// Trigger only a beam parameter mismatch
// Do not trip zero rate, unknown state, or debounce
PMPS_GVL.stCurrentBeamParameters := PMPS_GVL.cstFullBeam;
stBeamReq := PMPS_GVL.cstFullBeam;
stBeamReq.nTran := 0.5;
fbMiscFFO(
    fbArbiter:=fbArbiter,
    fbFFHWO:=fbFFHWO,
    stCurrentBeamReq:=stBeamReq,
    bKnownState:=TRUE,
    nTransitionID:=1,
);

fbFFHWO.EvaluateOutput();
AssertFalse(
    fbFFHWO.q_xFastFaultOut,
    'Did not fault with bad attenuator state',
);

TEST_FINISHED();
END_METHOD

METHOD TestDebounce
VAR_INST
    fbMiscFFO: FB_MiscStatesErrorFFO;
    fbArbiter: FB_Arbiter(5);
    fbFFHWO: FB_HardwareFFOutput := (bAutoReset := TRUE);
END_VAR
VAR
    nIter: DINT;
END_VAR

TEST('TestDebounce');

fbFFHWO.EvaluateOutput();
AssertTrue(
    fbFFHWO.q_xFastFaultOut,
    'Started with a fault prior to first FB run-through',
);
// Ask for full beam: there should be no faults of any kind
fbMiscFFO(
    fbArbiter:=fbArbiter,
    fbFFHWO:=fbFFHWO,
    stCurrentBeamReq:=PMPS_GVL.cstFullBeam,
    bKnownState:=TRUE,
    nTransitionID:=5,
);
fbFFHWO.EvaluateOutput();

AssertTrue(
    fbFFHWO.q_xFastFaultOut,
    'Started with a fault prior to trip checks',
);

// Trip and untrip the beam fast fault once, show no fault
TripUntrip(
    fbMiscFFO:=fbMiscFFO,
    fbArbiter:=fbArbiter,
    fbFFHWO:=fbFFHWO,
);
AssertTrue(
    fbFFHWO.q_xFastFaultOut,
    'Control group failed: one trip/untrip should not be enough to debounce',
);
// Trip and untrip the beam fast fault like 10 times, show fault
FOR nIter := 1 TO 10 DO
    TripUntrip(
        fbMiscFFO:=fbMiscFFO,
        fbArbiter:=fbArbiter,
        fbFFHWO:=fbFFHWO,
    );
END_FOR
AssertFalse(
    fbFFHWO.q_xFastFaultOut,
    'Debouncer failed to debounce',
);

TEST_FINISHED();
END_METHOD

METHOD TestTransitionState
VAR_INST
    fbMiscFFO: FB_MiscStatesErrorFFO;
    fbArbiter: FB_Arbiter(4);
    fbFFHWO: FB_HardwareFFOutput := (bAutoReset := TRUE);
END_VAR

TEST('TestTransitionState');

fbFFHWO.EvaluateOutput();
AssertTrue(
    fbFFHWO.q_xFastFaultOut,
    'Started with a fault',
);

// Trigger no faults, we're at an unknown state but it's a transition state
// Do not trip bad beam, zero rate, or debounce
fbArbiter.AddRequest(
    nReqID:=4,
    stReqBP:=PMPS_GVL.cstFullBeam,
    sDevName:='UnitTest',
);
PMPS_GVL.stCurrentBeamParameters := PMPS_GVL.cstFullBeam;
fbMiscFFO(
    fbArbiter:=fbArbiter,
    fbFFHWO:=fbFFHWO,
    stCurrentBeamReq:=PMPS_GVL.cstFullBeam,
    bKnownState:=FALSE,
    nTransitionID:=4,
);

fbFFHWO.EvaluateOutput();
AssertTrue(
    fbFFHWO.q_xFastFaultOut,
    'Faulted in unknown states even though we were moving normally',
);

TEST_FINISHED();
END_METHOD

METHOD TestUnknownState
VAR_INST
    fbMiscFFO: FB_MiscStatesErrorFFO;
    fbArbiter: FB_Arbiter(3);
    fbFFHWO: FB_HardwareFFOutput := (bAutoReset := TRUE);
END_VAR

TEST('TestUnknownState');

fbFFHWO.EvaluateOutput();
AssertTrue(
    fbFFHWO.q_xFastFaultOut,
    'Started with a fault',
);

// Trigger only an unknown states
// Do not trip bad beam, zero rate, or debounce
PMPS_GVL.stCurrentBeamParameters := PMPS_GVL.cstFullBeam;
fbMiscFFO(
    fbArbiter:=fbArbiter,
    fbFFHWO:=fbFFHWO,
    stCurrentBeamReq:=PMPS_GVL.cstFullBeam,
    bKnownState:=FALSE,
    nTransitionID:=3,
);

fbFFHWO.EvaluateOutput();
AssertFalse(
    fbFFHWO.q_xFastFaultOut,
    'Did not fault with unknown state',
);

TEST_FINISHED();
END_METHOD

METHOD TestZeroRate
VAR_INST
    fbMiscFFO: FB_MiscStatesErrorFFO;
    fbArbiter: FB_Arbiter(2);
    fbFFHWO: FB_HardwareFFOutput := (bAutoReset := TRUE);

    stNoBeam: ST_BeamParams;
END_VAR

TEST('TestBeamZeroRate');

fbFFHWO.EvaluateOutput();
AssertTrue(
    fbFFHWO.q_xFastFaultOut,
    'Started with a fault',
);

// Trigger only a zero rate
// Do not trip beam parameter mismatch, unknown state, or debounce
PMPS_GVL.stCurrentBeamParameters := stNoBeam;
fbMiscFFO(
    fbArbiter:=fbArbiter,
    fbFFHWO:=fbFFHWO,
    stCurrentBeamReq:=PMPS_GVL.cst0RateBeam,
    bKnownState:=TRUE,
    nTransitionID:=2
);

fbFFHWO.EvaluateOutput();
AssertFalse(
    fbFFHWO.q_xFastFaultOut,
    'Did not fault with zero rate',
);

TEST_FINISHED();
END_METHOD

METHOD TripUntrip
VAR_IN_OUT
    fbMiscFFO: FB_MiscStatesErrorFFO;
    fbArbiter: FB_Arbiter;
    fbFFHWO: FB_HardwareFFOutput;
END_VAR
VAR
    stBeamReq: ST_BeamParams;
END_VAR

// Use anything other than 0 rate, which is its own check
stBeamReq := PMPS_GVL.cstFullBeam;
stBeamReq.nTran := 0.5;
// Trip: too much beam!
PMPS_GVL.stCurrentBeamParameters := PMPS_GVL.cstFullBeam;
fbMiscFFO(
    fbArbiter:=fbArbiter,
    fbFFHWO:=fbFFHWO,
    stCurrentBeamReq:=stBeamReq,
    bKnownState:=TRUE,
    nTransitionID:=5,
);
fbFFHWO.EvaluateOutput();

// Untrip: correct beam!
PMPS_GVL.stCurrentBeamParameters := stBeamReq;
fbMiscFFO(
    fbArbiter:=fbArbiter,
    fbFFHWO:=fbFFHWO,
    stCurrentBeamReq:=stBeamReq,
    bKnownState:=TRUE,
    nTransitionID:=5,
);
fbFFHWO.EvaluateOutput();
END_METHOD

END_FUNCTION_BLOCK

// ---- POUs/Motion/PMPS/FB_MiscStatesErrorFFO.TcPOU
FUNCTION_BLOCK FB_MiscStatesErrorFFO
(*
    A catch-all for miscellaneous state FFOs that are not better organized elsewhere.
    Contains the following fast faults:
    - ffBeamParamsOK: trip the beam if the beam parameters are not safe enough for our current (known) state
    - ffZeroRate: trip the beam if we've asked for zero rate (as a shortcut)
    - ffUnknown: trip the beam if we're at an unknown state and our transition id is not asserted.
    - ffDebounce: trip the beam (no autoreset) if ffBeamParamsOK fast faults fault on and off multiple times too quickly.
      This solves an issue where ffBeamParamsOK might solve its own problem and creating a blinking fast fault issue.

    The inputs are mostly outputs of non-pmps function blocks and heavily-reused info like state details.
*)
VAR_IN_OUT
    // The arbiter to request beam states from
    fbArbiter: FB_Arbiter;
    // The fast fault output to fault to
    fbFFHWO: FB_HardwareFFOutput;
END_VAR
VAR_INPUT
    // A name to link to these fast faults
    sDeviceName: STRING;
    // Current requested beam details: either a known state or the transition beam
    stCurrentBeamReq: ST_BeamParams;
    // TRUE if we're at a known state (doesn't matter which)
    bKnownState: BOOL;
    // Lookup ID of the transition beam
    nTransitionID: DWORD;
    // Set me true to prevent any ffos from occuring
    bMaintenanceMode : BOOL;
END_VAR
VAR_OUTPUT
END_VAR
VAR CONSTANT
    // Number of consecutive trips before we debounce
    nMaxTrips: UINT := 5;
    // Decrease trip count by 1 after this much time has passed
    tTripReset: TIME := T#1s;
END_VAR
VAR
    // If the beam parameters are wrong, it is a fault! This encompasses all unknown arbiter-related errors.
    ffBeamParamsOk: FB_FastFault;
    // If we asked for zero rate (NC or SC) then we can cut the beam early. This is somewhat redundant.
    ffZeroRate: FB_FastFault;
    // Trip the beam for unknown state
    ffUnknown: FB_FastFault;
    // Trip the beam (no autoreset) if ffBeamParamsOK faults/resets multiple times too quickly.
    ffDebounce: FB_FastFault;

    // Number of consecutive trips so far
    nTripCount: UINT;
    // Increase by 1 whenever there is a fault (rising edge)
    ftTripCount: F_TRIG;
    // Decrease trip count by 1 each timeout
    tonTripCount: TON;
    // TRUE on only the first cycle
    bFirstCycle: BOOL := TRUE;
END_VAR


ffBeamParamsOk(
    i_xOK:=F_SafeBPCompare(PMPS_GVL.stCurrentBeamParameters, stCurrentBeamReq) OR bMaintenanceMode,
    i_xAutoReset:=TRUE,
    i_DevName:=sDeviceName,
    i_Desc:='Beam parameter mismatch',
    i_TypeCode:=E_MotionFFType.BP_MISMATCH,
    io_fbFFHWO:=fbFFHWO);

CASE PMPS_GVL.stCurrentBeamParameters.nMachineMode OF
    // NC mode
    1: ffZeroRate.i_xOK := stCurrentBeamReq.nRate > 0;
    // SC mode
    2: ffZeroRate.i_xOK := stCurrentBeamReq.nBCRange > 0;
ELSE
    // Ambiguous or new mode
    ffZeroRate.i_xOK := stCurrentBeamReq.nRate > 0 AND stCurrentBeamReq.nBCRange > 0;
END_CASE

ffZeroRate.i_xOK := ffZeroRate.i_xOK OR bMaintenanceMode;

ffZeroRate(
    i_xAutoReset := TRUE,
    i_DevName := sDeviceName,
    i_Desc := 'Device requesting zero rate',
    i_TypeCode := E_MotionFFType.ZERO_RATE,
    io_fbFFHWO := fbFFHWO,
);

ffUnknown(
    i_xOK := bknownState OR fbArbiter.CheckRequestInPool(nReqID:=nTransitionID) OR bMaintenanceMode,
    i_xAutoReset := TRUE,
    i_DevName := sDeviceName,
    i_Desc := 'Unknown position between moves',
    i_TypeCode := E_MotionFFType.NOT_A_STATE,
    io_fbFFHWO := fbFFHWO,
);

ftTripCount(CLK:=ffBeamParamsOk.i_xOK);

IF ftTripCount.Q THEN
    nTripCount := MIN(nTripCount + 1, 5);
END_IF

tonTripCount(
    IN:=NOT tonTripCount.Q,
    PT:=tTripReset,
);
IF tonTripCount.Q AND nTripCount > 0 THEN
    nTripCount := nTripCount - 1;
END_IF

// This is required for non-autoresetting FBs to come up in a beam permitted state
ffDebounce.i_xReset := bFirstCycle OR nTripCount=0;
ffDebounce(
    i_xOK := nTripCount < 5 OR bMaintenanceMode,
    i_DevName := sDeviceName,
    i_Desc := 'Tripped beam parameter mismatch off/on too many times, hold off',
    i_TypeCode := E_MotionFFType.TOO_MANY_TRIPS,
    io_fbFFHWO := fbFFHWO,
);
bFirstCycle := FALSE;

END_FUNCTION_BLOCK

// ---- Tests/FB_MotionBPTM_Test.TcPOU
FUNCTION_BLOCK FB_MotionBPTM_Test EXTENDS TcUnit.FB_TestSuite
(*
    Test the functionality of the motion bptm,
    Which is just a bptm wrapped up with a set of n motors.
    We're basically just making sure that we push the done button at the appropriate time.
    Direct tests of BPTM itself are reserved for the pmps library.

    The BPTM takes care of these executions across multiple cycles,
    so these tests must implement timeouts.
*)
VAR
    astMotionStage: ARRAY[1..MotionConstants.MAX_STATE_MOTORS] OF ST_MotionStage;
    stGoal1: ST_DbStateParams;
    stGoal2: ST_DbStateParams;
    stTrans: ST_DbStateParams;
    stNoBeam: ST_BeamParams;
END_VAR


stGoal1.stBeamParams := PMPS_GVL.cstFullBeam;
stGoal1.nRequestAssertionID := 1;
stGoal1.sPmpsState := 'stGoal1';
stGoal2.stBeamParams := PMPS_GVL.cstFullBeam;
stGoal2.stBeamParams.nTran := 0.5;
stGoal2.nRequestAssertionID := 2;
stGoal2.sPmpsState := 'stGoal2';
stTrans.stBeamParams := PMPS_GVL.cst0RateBeam;
stTrans.nRequestAssertionID := 3;
stTrans.sPmpsState := 'stTrans';

// Just put a blanket global no beam so these won't wait for any changes ever
PMPS_GVL.stCurrentBeamParameters := stNoBeam;
TestInit();
Test3dMove();
TestNoMove();
TestCount();
TestToggle();

METHOD AssertInPool
VAR_IN_OUT
    fbArbiter: FB_Arbiter;
    stDbStateParams: ST_DbStateParams;
END_VAR
VAR_INPUT
    bInPool: BOOL;
    sContext: STRING;
END_VAR

IF bInPool THEN
    AssertTrue(
        fbArbiter.CheckRequestInPool(stDbStateParams.nRequestAssertionID),
        CONCAT(CONCAT(stDbStateParams.sPmpsState, ' Beam parameters were not in the pool '), sContext),
    );
ELSE
    AssertFalse(
        fbArbiter.CheckRequestInPool(stDbStateParams.nRequestAssertionID),
        CONCAT(CONCAT(stDbStateParams.sPmpsState, ' Beam parameters unexpectedly found in the pool '), sContext),
    );
END_IF
END_METHOD

METHOD SetMotorDone
VAR_INPUT
END_VAR

// Force post-move state
astMotionStage[1].bBusy := FALSE;
astMotionStage[1].bDone := TRUE;
astMotionStage[2].bBusy := FALSE;
astMotionStage[2].bDone := TRUE;
astMotionStage[3].bBusy := FALSE;
astMotionStage[3].bDone := TRUE;
END_METHOD

METHOD SetMotorMoving
VAR_INPUT
END_VAR

// Force a moving but not done state
astMotionStage[1].bBusy := TRUE;
astMotionStage[1].bDone := FALSE;
astMotionStage[2].bBusy := TRUE;
astMotionStage[2].bDone := FALSE;
astMotionStage[3].bBusy := TRUE;
astMotionStage[3].bDone := FALSE;
END_METHOD

METHOD SetMotorStartup
VAR_INPUT
END_VAR

// Force some sort of default looking state
astMotionStage[1].bBusy := FALSE;
astMotionStage[1].bDone := FALSE;
astMotionStage[2].bBusy := FALSE;
astMotionStage[2].bDone := FALSE;
astMotionStage[3].bBusy := FALSE;
astMotionStage[3].bDone := FALSE;
END_METHOD

METHOD Test3dMove : BOOL
(*
    Can we safely do a 3d move?
*)
VAR_INST
    fbBptm: FB_MotionBPTM;
    fbArbiter: FB_Arbiter(2);
    fbFFHWO: FB_HardwareFFOutput := (bAutoReset := TRUE);
    fbSubSysIO : FB_DummyArbIO;

    nState: UINT;
    tonTimer: TON;
END_VAR

TEST('Test3DMove');

tonTimer(
    IN:=TRUE,
    PT:=T#5s,
);
IF tonTimer.Q THEN
    nState := 4;
END_IF

CASE nState OF
    0:
        // Establish baseline at Goal1
        SetMotorStartup();
        fbBptm(
            astMotionStage:=astMotionStage,
            fbArbiter:=fbArbiter,
            fbFFHWO:=fbFFHWO,
            stGoalParams:=stGoal1,
            stTransParams:=stTrans,
            nActiveMotorCount:=3,
            bEnable:=TRUE,
            bAtState:=TRUE,
        );
        IF fbBptm.bDone THEN
            nState := 1;
        END_IF
    1:
        // Request a move
        SetMotorStartup();
        fbBptm(
            astMotionStage:=astMotionStage,
            fbArbiter:=fbArbiter,
            fbFFHWO:=fbFFHWO,
            stGoalParams:=stGoal2,
            stTransParams:=stTrans,
            nActiveMotorCount:=3,
            bEnable:=TRUE,
            bAtState:=FALSE,
        );
        IF fbBptm.bTransitionAuthorized THEN
            // We should have transition and goal 2 asserts in
            AssertInPool(fbArbiter, stGoal1, FALSE, 'with trans auth');
            AssertInPool(fbArbiter, stGoal2, TRUE, 'with trans auth');
            AssertInPool(fbArbiter, stTrans, TRUE, 'with trans auth');
            nState := 2;
        END_IF
    2:
        // Simulate a move
        SetMotorMoving();
        fbBptm(
            astMotionStage:=astMotionStage,
            fbArbiter:=fbArbiter,
            fbFFHWO:=fbFFHWO,
            stGoalParams:=stGoal2,
            stTransParams:=stTrans,
            nActiveMotorCount:=3,
            bEnable:=TRUE,
            bAtState:=FALSE,
        );
        // Same situation as before
        AssertInPool(fbArbiter, stGoal1, FALSE, 'after move started');
        AssertInPool(fbArbiter, stGoal2, TRUE, 'after move started');
        AssertInPool(fbArbiter, stTrans, TRUE, 'after move started');
        nState := 3;
    3:
        // Move is done
        SetMotorDone();
        fbBptm(
            astMotionStage:=astMotionStage,
            fbArbiter:=fbArbiter,
            fbFFHWO:=fbFFHWO,
            stGoalParams:=stGoal2,
            stTransParams:=stTrans,
            nActiveMotorCount:=3,
            bEnable:=TRUE,
            bAtState:=TRUE,
        );
        IF fbBptm.bDone THEN
            // Dropped the transition assert
            AssertInPool(fbArbiter, stGoal1, FALSE, 'with move complete');
            AssertInPool(fbArbiter, stGoal2, TRUE, 'with move complete');
            AssertInPool(fbArbiter, stTrans, FALSE, 'with move complete');
            nState := 4;
        END_IF
    4:
        AssertFalse(
            tonTimer.Q,
            'Timeout in test',
        );
        TEST_FINISHED();
END_CASE

fbSubSysIO(
    LA:=fbArbiter,
    FFO:=fbFFHWO,
);
END_METHOD

METHOD TestCount
(*
    FB Should just error out if we forgot to give a count
*)
VAR_INST
    fbBptm: FB_MotionBPTM;
    fbArbiter: FB_Arbiter(1);
    fbFFHWO: FB_HardwareFFOutput := (bAutoReset := TRUE);

    tonWait: TON;
END_VAR
TEST('TestCount');

SetMotorStartup();
fbBptm(
    astMotionStage:=astMotionStage,
    fbArbiter:=fbArbiter,
    fbFFHWO:=fbFFHWO,
    stGoalParams:=stGoal1,
    stTransParams:=stTrans,
    bEnable:=True,
    bAtState:=True,
);
AssertTrue(
    fbBptm.bMotorCountError,
    'Did not properly error on missing motor count',
);

tonWait(
    IN:=TRUE,
    PT:=T#1s,
);
IF tonWait.Q THEN
    // Should have no arbiter activity at all
    AssertInPool(fbArbiter, stGoal1, FALSE, 'with bad count');
    AssertInPool(fbArbiter, stGoal2, FALSE, 'with bad count');
    AssertInPool(fbArbiter, stTrans, FALSE, 'with bad count');

    TEST_FINISHED();
END_IF
END_METHOD

METHOD TestInit : BOOL
(*
    If we initialize with still motors, do we get an arbiter request at the current goal? Hopefully we do.
*)
VAR_INST
    fbBptm: FB_MotionBPTM;
    fbArbiter: FB_Arbiter(1);
    fbFFHWO: FB_HardwareFFOutput := (bAutoReset := TRUE);
    fbSubSysIO : FB_DummyArbIO;

    tonTimer: TON;
END_VAR

TEST('TestInit');

SetMotorStartup();
fbBptm(
    astMotionStage:=astMotionStage,
    fbArbiter:=fbArbiter,
    fbFFHWO:=fbFFHWO,
    stGoalParams:=stGoal1,
    stTransParams:=stTrans,
    nActiveMotorCount:=3,
    bEnable:=True,
    bAtState:=True,
);
fbSubSysIO(
    LA:=fbArbiter,
    FFO:=fbFFHWO,
);

tonTimer(
    IN:=TRUE,
    PT:=T#5s,
);
IF tonTimer.Q OR fbBptm.bDone THEN
    AssertFalse(
        tonTimer.Q,
        'Timeout in test',
    );
    // We should have a request in the pool for goal 1 but not for transition
    // If no request are in the pool, we may come up in a no protection state!
    // If both requests are in the pool, we may come up in a too much blocking beam state!
    AssertInPool(fbArbiter, stGoal1, TRUE, 'at startup');
    AssertInPool(fbArbiter, stTrans, FALSE, 'at startup');

    TEST_FINISHED();
END_IF
END_METHOD

METHOD TestNoMove
(*
    In place transitions should work at startup and also at done positions.
*)
VAR_INST
    fbBptm: FB_MotionBPTM;
    fbArbiter: FB_Arbiter(1);
    fbFFHWO: FB_HardwareFFOutput := (bAutoReset := TRUE);
    fbSubSysIO : FB_DummyArbIO;

    nState: UINT;
    tonTimer: TON;
END_VAR

TEST('TestNoMove');

tonTimer(
    IN:=TRUE,
    PT:=T#5s,
);
IF tonTimer.Q THEN
    nState := 3;
END_IF

CASE nState OF
    0:
        SetMotorStartup();
        fbBptm(
            astMotionStage:=astMotionStage,
            fbArbiter:=fbArbiter,
            fbFFHWO:=fbFFHWO,
            stGoalParams:=stGoal1,
            stTransParams:=stTrans,
            nActiveMotorCount:=3,
            bEnable:=True,
            bAtState:=True,
        );
        IF fbBptm.bDone THEN
            nState := 1;
        END_IF
    1:
        SetMotorStartup();
        // NOTE: we kept bAtState TRUE the whole time, so this should be a completed in-place transition
        fbBptm(
            astMotionStage:=astMotionStage,
            fbArbiter:=fbArbiter,
            fbFFHWO:=fbFFHWO,
            stGoalParams:=stGoal2,
            stTransParams:=stTrans,
            nActiveMotorCount:=3,
            bEnable:=True,
            bAtState:=True,
        );
        IF fbBptm.bDone THEN
            // Only Goal2 should be in the pool
            AssertInPool(fbArbiter, stGoal1, FALSE, 'after switching goals (1)');
            AssertInPool(fbArbiter, stGoal2, TRUE, 'after switching goals (1)');
            AssertInPool(fbArbiter, stTrans, FALSE, 'after switching goals (1)');
            nState := 2;
        END_IF
    2:
        // Repeat from a done position!
        SetMotorDone();
        fbBptm(
            astMotionStage:=astMotionStage,
            fbArbiter:=fbArbiter,
            fbFFHWO:=fbFFHWO,
            stGoalParams:=stGoal1,
            stTransParams:=stTrans,
            nActiveMotorCount:=3,
            bEnable:=True,
            bAtState:=True,
        );
        IF fbBptm.bDone THEN
            // Only Goal1 should be in the pool
            AssertInPool(fbArbiter, stGoal1, TRUE, 'after switching goals (2)');
            AssertInPool(fbArbiter, stGoal2, FALSE, 'after switching goals (2)');
            AssertInPool(fbArbiter, stTrans, FALSE, 'after switching goals (2)');
            nState := 3;
        END_IF
    3:
        AssertFalse(
            tonTimer.Q,
            'Timeout in test',
        );
        TEST_FINISHED();
END_CASE

fbSubSysIO(
    LA:=fbArbiter,
    FFO:=fbFFHWO,
);
END_METHOD

METHOD TestToggle
(*
    Arbitration requests should be added to pool even if there is no transition, as case which occurs
    when a BeamParameterTransitionManager is not processed for at least one cycle without changing states
    and then reprocessed, usually when arbitration is temporarily disabled to deal with unrelated faults.
*)
VAR_INST
    fbBptm: FB_MotionBPTM;
    fbArbiter: FB_Arbiter(1);
    fbFFHWO: FB_HardwareFFOutput := (bAutoReset := TRUE);
    fbSubSysIO : FB_DummyArbIO;

    nState: UINT;
    tonTimer: TON;
END_VAR

TEST('TestToggle');

tonTimer(
    IN:=TRUE,
    PT:=T#5s,
);
IF tonTimer.Q THEN
    nState := 4;
END_IF

CASE nState OF
    0:
        SetMotorStartup();
        fbBptm(
            astMotionStage:=astMotionStage,
            fbArbiter:=fbArbiter,
            fbFFHWO:=fbFFHWO,
            stGoalParams:=stGoal1,
            stTransParams:=stTrans,
            nActiveMotorCount:=3,
            bEnable:=True,
            bAtState:=True,
        );
        IF fbBptm.bDone THEN
            nState := 1;
        END_IF
    1:
        SetMotorStartup();
        // NOTE: we kept bAtState TRUE the whole time, so this should be a completed in-place transition
        fbBptm(
            astMotionStage:=astMotionStage,
            fbArbiter:=fbArbiter,
            fbFFHWO:=fbFFHWO,
            stGoalParams:=stGoal2,
            stTransParams:=stTrans,
            nActiveMotorCount:=3,
            bEnable:=True,
            bAtState:=True,
        );
        IF fbBptm.bDone THEN
            // Only Goal2 should be in the pool
            AssertInPool(fbArbiter, stGoal1, FALSE, 'after switching goals (1)');
            AssertInPool(fbArbiter, stGoal2, TRUE, 'after switching goals (1)');
            AssertInPool(fbArbiter, stTrans, FALSE, 'after switching goals (1)');
            nState := 2;
        END_IF
    2:
        // Run disabled
        SetMotorDone();
        fbBptm(
            astMotionStage:=astMotionStage,
            fbArbiter:=fbArbiter,
            fbFFHWO:=fbFFHWO,
            stGoalParams:=stGoal2,
            stTransParams:=stTrans,
            nActiveMotorCount:=3,
            bEnable:=False,
            bAtState:=True,
        );
        IF fbBptm.bDone THEN
            // Nothing should be in the pool
            AssertInPool(fbArbiter, stGoal1, FALSE, 'after switching goals (2)');
            AssertInPool(fbArbiter, stGoal2, FALSE, 'after switching goals (2)');
            AssertInPool(fbArbiter, stTrans, FALSE, 'after switching goals (2)');
            nState := 3;
        END_IF
    3:
        // Re-enable without changing goal
        fbBptm(
            astMotionStage:=astMotionStage,
            fbArbiter:=fbArbiter,
            fbFFHWO:=fbFFHWO,
            stGoalParams:=stGoal2,
            stTransParams:=stTrans,
            nActiveMotorCount:=3,
            bEnable:=True,
            bAtState:=True,
        );
        IF fbBptm.bDone THEN
            //  Goal2 should be back in the pool
            AssertInPool(fbArbiter, stGoal1, FALSE, 'after switching goals (2)');
            AssertInPool(fbArbiter, stGoal2, TRUE, 'after switching goals (2)');
            AssertInPool(fbArbiter, stTrans, FALSE, 'after switching goals (2)');
            nState := 4;
        END_IF
    4:
        AssertFalse(
            tonTimer.Q,
            'Timeout in test',
        );
        TEST_FINISHED();
END_CASE

fbSubSysIO(
    LA:=fbArbiter,
    FFO:=fbFFHWO,
);
END_METHOD

END_FUNCTION_BLOCK

// ---- POUs/Motion/PMPS/FB_MotionBPTM.TcPOU

FUNCTION_BLOCK FB_MotionBPTM
(*
    This function block handles the beam parameter transition manager for a group of motors moving together to a destination with shared beam state.
    stGoalParams and stTransParams are required arguments and must not share IDs with other state parameters in the PLC.

    This is a building block not intended for use outside of lcls-twincat-motion.
*)
VAR_IN_OUT
    // Array of motors that will move for this beam transition
    astMotionStage: ARRAY[1..MotionConstants.MAX_STATE_MOTORS] OF ST_MotionStage;
    // The arbiter to request beam states from
    fbArbiter: FB_Arbiter;
    // The fast fault output to fault to
    fbFFHWO: FB_HardwareFFOutput;
    // The parameters we want to transition to
    stGoalParams: ST_DbStateParams;
    // The parameters we want to use during the transition
    stTransParams: ST_DbStateParams;
END_VAR
VAR_INPUT
    // The number of motors we're actually using
    nActiveMotorCount: UINT;
    // Set to TRUE to use the BPTM, FALSE to stop using the BPTM.
    bEnable: BOOL;
    // TRUE if we're at the physical state that matches the goal parameters
    bAtState: BOOL;
    // A device name to use in the GUI
    sDeviceName: STRING;
    // How long to wait for parameters before timing out
    tArbiterTimeout: TIME := T#1s;
    // Whether to fault and move on timeout (TRUE) or to wait (FALSE)
    bMoveOnArbiterTimeout: BOOL := TRUE;
    // Set to TRUE when it is safe to reset the BPTM timeout fast fault, to reset it early.
    bResetBPTMTimeout: BOOL;
    // Set to TRUE to make the BPTM retry
    bRetry: BOOL;
END_VAR
VAR_OUTPUT
    // This becomes TRUE when the motors are allowed to move to their destinations.
    bTransitionAuthorized: BOOL;
    // This becomes TRUE once the full beam transition is done.
    bDone: BOOL;
    // TRUE if we're using a bad motor count
    bMotorCountError: BOOL;
END_VAR
VAR
    bptm: BeamParameterTransitionManager;
    bDoneMoving: BOOL;
    nPrevID: UDINT;
    nIndex: DINT;

    bInternalAuth: BOOL;
    bDoneResetQueued: BOOL;

    tonArbiter: TON;
    bArbiterTimeout: BOOL;
    ffBPTMTimeoutAndMove: FB_FastFault;
    ffBPTMError: FB_FastFault;
END_VAR


CheckCount();
IF NOT bMotorCountError THEN
    SetDoneMoving();
    IF bEnable THEN
        RunBPTM();
    END_IF
    HandleTimeout();
END_IF

ACTION CheckCount:

// Make sure the motor count is valid (positive, nonzero, less or equal to the max)
bMotorCountError S= nActiveMotorCount <= 0;
bMotorCountError S= nActiveMotorCount > MotionConstants.MAX_STATE_MOTORS;
END_ACTION

ACTION HandleTimeout:

// Measure the time that the bptm is busy
tonArbiter(
    IN:=bptm.bBusy,
    PT:=tArbiterTimeout,
    Q=>bArbiterTimeout,
);
bTransitionAuthorized := bInternalAuth OR (bArbiterTimeout AND bMoveOnArbiterTimeout);

// Trip the beam for BPTM timeouts if we want to move
// Only reset at safe beam OR at no bptm errors (some other FF should catch additional issues)
ffBPTMTimeoutAndMove.i_xOK := NOT (bArbiterTimeout AND bMoveOnArbiterTimeout) OR (NOT THIS^.bEnable);
ffBPTMTimeoutAndMove.i_xReset S= bResetBPTMTimeout OR (bptm.bDone AND NOT bptm.bError);
ffBPTMTimeoutAndMove.i_xReset R= NOT ffBPTMTimeoutAndMove.i_xOK;
ffBPTMTimeoutAndMove.i_xReset := ffBPTMTimeoutAndMove.i_xReset OR NOT bEnable;
ffBPTMTimeoutAndMove(
    i_DevName := sDeviceName,
    i_Desc := 'BPTM Timeout',
    i_TypeCode := E_MotionFFType.BPTM_TIMEOUT,
    io_fbFFHWO := fbFFHWO,
);
END_ACTION

ACTION RunBPTM:

bptm(
    fbArbiter:=fbArbiter,
    i_sDeviceName:=sDeviceName,
    i_TransitionAssertionID:=stTransParams.nRequestAssertionID,
    i_stTransitionAssertion:=stTransParams.stBeamParams,
    i_nRequestedAssertionID:=stGoalParams.nRequestAssertionID,
    i_stRequestedAssertion:=stGoalParams.stBeamParams,
    i_xDoneMoving:=bDoneMoving AND bAtState,
    stCurrentBeamParameters:=PMPS_GVL.stCurrentBeamParameters,
    bRetry:=bRetry,
    q_xTransitionAuthorized=>bInternalAuth,
    bDone=>bDone,
);

// Trip the beam for BPTM Errors
ffBPTMError.i_xOK := (NOT bptm.bError) OR NOT THIS^.bEnable;
ffBPTMError.i_xReset S= bptm.bDone AND ffBPTMError.i_xOK;
ffBPTMError.i_xReset R= NOT ffBPTMError.i_xOK;
ffBPTMError(
    i_DevName := sDeviceName,
    i_Desc := 'BPTM error, state transition failed',
    i_TypeCode := E_MotionFFType.BPTM_ERROR,
    io_fbFFHWO := fbFFHWO,
);
END_ACTION

ACTION SetDoneMoving:

// Set bDoneMoving if all the motors are done
bDoneMoving := TRUE;
FOR nIndex := 1 TO nActiveMotorCount DO
    bDoneMoving := bDoneMoving AND NOT astMotionStage[nIndex].bBusy AND NOT astMotionStage[nIndex].bExecute;
END_FOR
// Reset bDoneMoving if the goal has changed to reset bptm's motor done for an in-place transition
// This allows us to change to a new beam state without requiring a motor state change
// BPTM only checks for this "done" transition after the transition has been authorized, so we may need to wait
bDoneResetQueued S= nPrevID <> stGoalParams.nRequestAssertionID;
bDoneMoving R= bDoneResetQueued AND bptm.q_xTransitionAuthorized;
bDoneResetQueued R= bptm.q_xTransitionAuthorized;
nPrevID := stGoalParams.nRequestAssertionID;
END_ACTION

END_FUNCTION_BLOCK

// ---- Tests/FB_MotionClearAsserts_Test.TcPOU
FUNCTION_BLOCK FB_MotionClearAsserts_Test EXTENDS TcUnit.FB_TestSuite
VAR
END_VAR


TestBasic();

METHOD TestBasic
VAR
    nIter: UINT;
END_VAR
VAR_INST
    fbClear: FB_MotionClearAsserts;
    astDbStateParams: ARRAY[0..GeneralConstants.MAX_STATES] OF ST_DbStateParams;
    fbArbiter: FB_Arbiter(1);
END_VAR

TEST('TestBasic');

FOR nIter := 0 TO GeneralConstants.MAX_STATES DO
    astDbStateParams[nIter].nRequestAssertionID := 100 + nIter;
    fbArbiter.AddRequest(
        nReqID:=100 + nIter,
        stReqBP:=PMPS_GVL.cstFullBeam,
        sDevName:='UnitTest',
    );
END_FOR

FOR nIter := 0 TO GeneralConstants.MAX_STATES DO
    AssertTrue(
        fbArbiter.CheckRequestInPool(100 + nIter),
        CONCAT(CONCAT('State ', UDINT_TO_STRING(nIter)), ' was not in the pool'),
    );
END_FOR

fbClear(
    astDbStateParams:=astDbStateParams,
    fbArbiter:=fbArbiter,
    bExecute:=TRUE,
);

FOR nIter := 0 TO GeneralConstants.MAX_STATES DO
    AssertFalse(
        fbArbiter.CheckRequestInPool(100 + nIter),
        CONCAT(CONCAT('State ', UDINT_TO_STRING(nIter)), ' was not cleared from the pool'),
    );
END_FOR

TEST_FINISHED();
END_METHOD

END_FUNCTION_BLOCK

// ---- POUs/Motion/PMPS/FB_MotionClearAsserts.TcPOU
FUNCTION_BLOCK FB_MotionClearAsserts
(*
    Clear all of the PMPS asserts related to a states mover.
*)
VAR_IN_OUT
    // All states to deactivate: transition + the static position states
    astDbStateParams: ARRAY[0..GeneralConstants.MAX_STATES] OF ST_DbStateParams;
    // The arbiter who made the PMPS assert requests
    fbArbiter: FB_ARBITER;
END_VAR
VAR_INPUT
    // Clear asserts on rising edge
    bExecute: BOOL;
END_VAR
VAR_OUTPUT
END_VAR
VAR
    rtExec: R_TRIG;
    nIter: DINT;
END_VAR


rtExec(CLK:=bExecute);
IF rtExec.Q THEN
    FOR nIter := 0 TO GeneralConstants.MAX_STATES DO
        fbArbiter.RemoveRequest(astDbStateParams[nIter].nRequestAssertionID);
    END_FOR
END_IF

END_FUNCTION_BLOCK

// ---- Tests/FB_MotionReadPMPSDBND_Test.TcPOU
FUNCTION_BLOCK FB_MotionReadPMPSDBND_Test EXTENDS TcUnit.FB_TestSuite
(*
    We test the actual db read in the pmps lib
    Here, we test that the correct keys are ready for the read based on the inputs.

    The user submits a transition key and all of their ST_PositionState instances from all of their motors.
    Any subset of these instances can have lookup keys.

    If only one state at the index has a lookup key, use that key.
    If more than one state at the index has the same lookup key, use that key.
    If states at the same index have different keys, that's an error and a fast fault.
    If states at different indices have the same keys, that's an error and a fast fault.
*)
VAR
    astCorrectStates: ARRAY[1..GeneralConstants.MAX_STATES] OF ST_PositionState;
    astNonsenseStates: ARRAY[1..GeneralConstants.MAX_STATES] OF ST_PositionState;
    astDuplicatedStates: ARRAY[1..GeneralConstants.MAX_STATES] OF ST_PositionState;
    astHalfFullStates: ARRAY[1..GeneralConstants.MAX_STATES] OF ST_PositionState;
    nIter: UINT;
END_VAR


// Set up the state arrays that can be used in test methods
FOR nIter := 1 TO GeneralConstants.MAX_STATES DO
    astCorrectStates[nIter].stPMPS.sPmpsState := CONCAT('State', UINT_TO_STRING(nIter));
    astNonsenseStates[nIter].stPMPS.sPmpsState := CONCAT('asdf', UINT_TO_STRING(nIter));
    IF UINT_TO_BOOL(nIter MOD 2) THEN
        astDuplicatedStates[nIter].stPMPS.sPmpsState := 'State0';
    ELSE
        astDuplicatedStates[nIter].stPMPS.sPmpsState := 'State1';
    END_IF
    IF nIter <= GeneralConstants.MAX_STATES / 2 THEN
        astHalfFullStates[nIter].stPMPS.sPmpsState := CONCAT('State', UINT_TO_STRING(nIter));
    END_IF
END_FOR

TestSolo();
TestTrio();
TestNonsense();
TestDupe();
TestBackfill();
TestHalfFull();

METHOD TestBackfill
VAR_INST
    fbRead: FB_MotionReadPMPSDBND;
    astPositionState: ARRAY[1..MotionConstants.MAX_STATE_MOTORS] OF ARRAY[1..GeneralConstants.MAX_STATES] OF ST_PositionState;
    fbFFHWO: FB_HardwareFFOutput := (bAutoReset := TRUE);
    stDefaultBP: ST_DbStateParams;
END_VAR

TEST('TestBackfill');

astPositionState[1] := astCorrectStates;
// Pick a few parameters to drop in
astPositionState[1][3].stPMPS.stBeamParams.nRate := 999;
astPositionState[2][1].stPMPS.nRequestAssertionID := 777;
astPositionState[3][2].stPMPS.bBeamParamsLoaded := NOT stDefaultBP.bBeamParamsLoaded;
fbRead(
    astPositionState:=astPositionState,
    fbFFHWO:=fbFFHWO,
    sTransitionKey:='State0',
    sDeviceName:='TestBackfill',
);
// Everything should be cleared to the defaults: the library should let us know what params got loaded (none)
AssertEquals_UDINT(
    Expected:=stDefaultBP.stBeamParams.nRate,
    Actual:=astPositionState[1][3].stPMPS.stBeamParams.nRate,
    Message:='nRate of motor 1 state 3 not backfilled',
);
AssertEquals_UDINT(
    Expected:=stDefaultBP.nRequestAssertionID,
    Actual:=astPositionState[2][1].stPMPS.nRequestAssertionID,
    Message:='nRequestAssertionID of motor 2 state 3 not backfilled',
);
AssertEquals_BOOL(
    Expected:=stDefaultBP.bBeamParamsLoaded,
    Actual:=astPositionState[3][2].stPMPS.bBeamParamsLoaded,
    Message:='bBeamParamsLoaded of motor 3 state 2 not backfilled',
);

TEST_FINISHED();
END_METHOD

METHOD TestDupe
VAR_INST
    fbRead: FB_MotionReadPMPSDBND;
    astPositionState: ARRAY[1..MotionConstants.MAX_STATE_MOTORS] OF ARRAY[1..GeneralConstants.MAX_STATES] OF ST_PositionState;
    fbFFHWO: FB_HardwareFFOutput := (bAutoReset := TRUE);
END_VAR

TEST('TestDupe');

astPositionState[1] := astDuplicatedStates;
fbRead(
    astPositionState:=astPositionState,
    fbFFHWO:=fbFFHWO,
    sTransitionKey:='State0',
    sDeviceName:='TestTrio',
);
fbFFHWO.EvaluateOutput();

AssertTrue(
    fbRead.bError,
    'Should have had an error',
);
FOR nIter := 0 TO GeneralConstants.MAX_STATES DO
    AssertEquals_STRING(
        Expected:='',
        Actual:=fbRead.astDbStateParams[nIter].sPmpsState,
        Message:=CONCAT('Errored output should have had no state names: ', UINT_TO_STRING(nIter)),
    );
END_FOR

TEST_FINISHED();
END_METHOD

METHOD TestHalfFull
VAR_INST
    fbRead: FB_MotionReadPMPSDBND;
    astPositionState: ARRAY[1..MotionConstants.MAX_STATE_MOTORS] OF ARRAY[1..GeneralConstants.MAX_STATES] OF ST_PositionState;
    fbFFHWO: FB_HardwareFFOutput := (bAutoReset := TRUE);
END_VAR

TEST('TestHalfFull');

astPositionState[1] := astHalfFullStates;
fbRead(
    astPositionState:=astPositionState,
    fbFFHWO:=fbFFHWO,
    sTransitionKey:='State0',
    sDeviceName:='TestHalfFull',
);
fbFFHWO.EvaluateOutput();

AssertFalse(
    fbRead.bError,
    'Had an error',
);
AssertEquals_STRING(
    Expected:=fbRead.sTransitionKey,
    Actual:=fbRead.astDbStateParams[0].sPmpsState,
    Message:='Output did not have the correct transition state',
);
FOR nIter := 1 TO GeneralConstants.MAX_STATES / 2 DO
    AssertEquals_STRING(
        Expected:=astCorrectStates[nIter].stPMPS.sPmpsState,
        Actual:=fbRead.astDbStateParams[nIter].sPmpsState,
        Message:=CONCAT('Output did not have the correct position state: ', UINT_TO_STRING(nIter)),
    );
END_FOR

TEST_FINISHED();
END_METHOD

METHOD TestNonsense
VAR_INST
    fbRead: FB_MotionReadPMPSDBND;
    astPositionState: ARRAY[1..MotionConstants.MAX_STATE_MOTORS] OF ARRAY[1..GeneralConstants.MAX_STATES] OF ST_PositionState;
    fbFFHWO: FB_HardwareFFOutput := (bAutoReset := TRUE);
END_VAR

TEST('TestNonsense');

astPositionState[1] := astCorrectStates;
astPositionState[2] := astNonsenseStates;
fbRead(
    astPositionState:=astPositionState,
    fbFFHWO:=fbFFHWO,
    sTransitionKey:='State0',
    sDeviceName:='TestTrio',
);
fbFFHWO.EvaluateOutput();

AssertTrue(
    fbRead.bError,
    'Should have had an error',
);
// Only the transition state should be spared from the nonsense
AssertEquals_STRING(
    Expected:='State0',
    Actual:=fbRead.astDbStateParams[0].sPmpsState,
    Message:='Transition state should be OK',
);
FOR nIter := 1 TO GeneralConstants.MAX_STATES DO
    AssertEquals_STRING(
        Expected:='',
        Actual:=fbRead.astDbStateParams[nIter].sPmpsState,
        Message:=CONCAT('Errored output should have had no state names: ', UINT_TO_STRING(nIter)),
    );
END_FOR

TEST_FINISHED();
END_METHOD

METHOD TestSolo
VAR_INST
    fbRead: FB_MotionReadPMPSDBND;
    astPositionState: ARRAY[1..MotionConstants.MAX_STATE_MOTORS] OF ARRAY[1..GeneralConstants.MAX_STATES] OF ST_PositionState;
    fbFFHWO: FB_HardwareFFOutput := (bAutoReset := TRUE);
END_VAR

TEST('TestSolo');

astPositionState[1] := astCorrectStates;
fbRead(
    astPositionState:=astPositionState,
    fbFFHWO:=fbFFHWO,
    sTransitionKey:='State0',
    sDeviceName:='TestSolo',
);
fbFFHWO.EvaluateOutput();

AssertFalse(
    fbRead.bError,
    'Had an error',
);
AssertEquals_STRING(
    Expected:=fbRead.sTransitionKey,
    Actual:=fbRead.astDbStateParams[0].sPmpsState,
    Message:='Output did not have the correct transition state',
);
FOR nIter := 1 TO GeneralConstants.MAX_STATES DO
    AssertEquals_STRING(
        Expected:=astCorrectStates[nIter].stPMPS.sPmpsState,
        Actual:=fbRead.astDbStateParams[nIter].sPmpsState,
        Message:=CONCAT('Output did not have the correct position state: ', UINT_TO_STRING(nIter)),
    );
END_FOR

TEST_FINISHED();
END_METHOD

METHOD TestTrio
VAR_INST
    fbRead: FB_MotionReadPMPSDBND;
    astPositionState: ARRAY[1..MotionConstants.MAX_STATE_MOTORS] OF ARRAY[1..GeneralConstants.MAX_STATES] OF ST_PositionState;
    fbFFHWO: FB_HardwareFFOutput := (bAutoReset := TRUE);
END_VAR

TEST('TestTrio');

astPositionState[1] := astCorrectStates;
astPositionState[2] := astCorrectStates;
astPositionState[3] := astCorrectStates;
fbRead(
    astPositionState:=astPositionState,
    fbFFHWO:=fbFFHWO,
    sTransitionKey:='State0',
    sDeviceName:='TestTrio',
);
fbFFHWO.EvaluateOutput();

AssertFalse(
    fbRead.bError,
    'Had an error',
);
AssertEquals_STRING(
    Expected:=fbRead.sTransitionKey,
    Actual:=fbRead.astDbStateParams[0].sPmpsState,
    Message:='Output did not have the correct transition state',
);
FOR nIter := 1 TO GeneralConstants.MAX_STATES DO
    AssertEquals_STRING(
        Expected:=astCorrectStates[nIter].stPMPS.sPmpsState,
        Actual:=fbRead.astDbStateParams[nIter].sPmpsState,
        Message:=CONCAT('Output did not have the correct position state: ', UINT_TO_STRING(nIter)),
    );
END_FOR

TEST_FINISHED();
END_METHOD

END_FUNCTION_BLOCK

// ---- POUs/Motion/PMPS/FB_MotionReadPMPSDBND.TcPOU
FUNCTION_BLOCK FB_MotionReadPMPSDBND
(*
    When we read the JSON PMPS database file, update the lookup parameters for one state mover.
    It is a building block not meant for use outside of lcls-twincat-motion.

    This is intended to support one N-dimensional state motion function block.
    The keys for the database lookup can be set on any of the motor's position states.
    Each of them have an allocated state.stPMPS.sPmpsState STRING parameter.
    If there is a conflict and two of the motors disagree on parameter lookups, that will
    be a fast fault.

    When the global JSON read function block is no longer busy and has no errors,
    we will assume that the file has been read and we will update the parameters here.

    This will also re-read in the event that the input position state keys change in any way,
    provided that we've read once before.
*)
VAR_IN_OUT
    // Each motor's respective position states along its direction. These will not be modified.
    astPositionState: ARRAY[1..MotionConstants.MAX_STATE_MOTORS] OF ARRAY[1..GeneralConstants.MAX_STATES] OF ST_PositionState;
    // Hardware output to fault to if there is a problem.
    fbFFHWO: FB_HardwareFFOutput;
END_VAR
VAR_INPUT
    // The database lookup key for the transition state. This has no corresponding ST_PositionState.
    sTransitionKey: STRING;
    // A name to use for fast faults, etc.
    sDeviceName: STRING;
    // For debug: set this to TRUE in online mode to read the database immediately.
    bReadNow: BOOL;
    // Set this to FALSE to load PMPS parameters locally
    bUsePmpsDB: BOOL := TRUE;
    // Local PMPSDB parameteres
    astManualDbStateParams:  ARRAY[0..GeneralConstants.MAX_STATES] OF ST_DbStateParams;
END_VAR
VAR_OUTPUT
    // The raw lookup results from this FB. Index 0 is the transition beam, the rest of the indices match the state positions.
    astDbStateParams: ARRAY[0..GeneralConstants.MAX_STATES] OF ST_DbStateParams;
    // TRUE if we've had at least one successful read.
    bFirstReadDone: BOOL;
    // This will be set to TRUE if there was an error reading from the database.
    bError: BOOL;
END_VAR
VAR
    ffError: FB_FastFault;
    fbReadPmpsDb: FB_JsonDocToSafeBP;
    ftDbBusy: F_TRIG;
    ftRead: F_TRIG;
    bReadPmpsDb: BOOL;
    nIterMotor: DINT;
    nIterState: DINT;
    nIterState2: DINT;
    sLoopNewKey: STRING;
    sLoopPrevKey: STRING;
    abStateError: ARRAY[0..GeneralConstants.MAX_STATES] OF BOOL;
    asLookupKeys: ARRAY[0..GeneralConstants.MAX_STATES] OF STRING;
    asPrevLookupKeys: ARRAY[0..GeneralConstants.MAX_STATES] OF STRING;
    bNewKeys: BOOL;
    sTempBackfill: STRING;
END_VAR

IF bUsePmpsDB THEN
    SelectLookupKeys();
    ReadDatabase();
    RunFastFaults();
    BackfillInfo();
ELSE
    astDbStateParams:=astManualDbStateParams;
END_IF

ACTION BackfillInfo:

// Put the results of the PMPS lookup back to the motion states
// This is purely for debugging purposes, as only the astDbStateParams output is used by the libraries.

// Copy everything except for the lookup key: avoid clobbering the user's original keys
// Do it this way instead of one element at a time to be forwards-compatible with any future additions to the db struct
FOR nIterState := 1 TO GeneralConstants.MAX_STATES DO
    FOR nIterMotor := 1 TO MotionConstants.MAX_STATE_MOTORS DO
        sTempBackfill := astPositionState[nIterMotor][nIterState].stPMPS.sPmpsState;
        astPositionState[nIterMotor][nIterState].stPMPS := astDbStateParams[nIterState];
        astPositionState[nIterMotor][nIterState].stPMPS.sPmpsState := sTempBackfill;
    END_FOR
END_FOR
END_ACTION

ACTION ReadDatabase:

// Read the database at the right timing
ftDbBusy(CLK:=MOTION_GVL.fbPmpsFileReader.bBusy);
IF ftDbBusy.Q THEN
    bReadPmpsDb S= NOT MOTION_GVL.fbPmpsFileReader.bError;
END_IF

bReadPmpsDb S= bFirstReadDone AND bNewKeys;
bReadPmpsDb S= bReadNow;
bReadNow := FALSE;

fbReadPmpsDb(
    bExecute:=bReadPmpsDb,
    jsonDoc:=PMPS_GVL.BP_jsonDoc,
    sDeviceName:=sDeviceName,
    io_fbFFHWO:=fbFFHWO,
    arrStates:=astDbStateParams,
);
bReadPmpsDb R= NOT fbReadPmpsDb.bBusy;

ftRead(CLK:=fbReadPmpsDb.bBusy);
bFirstReadDone S= ftRead.Q AND NOT fbReadPmpsDb.bError;
END_ACTION

ACTION RunFastFaults:

ffError(
    i_xOK:=NOT bError,
    i_xAutoReset:=TRUE,
    i_DevName:=sDeviceName,
    i_Desc:='Programmer error selecting state names in ND motion FB',
    i_TypeCode:=E_MotionFFType.INTERNAL_ERROR,
    io_fbFFHWO:=fbFFHWO,
);
END_ACTION

ACTION SelectLookupKeys:

// Fill the lookup key information in astDbStateParams based on the strings from astPositionState and sTransitionKey.

// Start by emptying any pre-existing values
FOR nIterState := 0 TO GeneralConstants.MAX_STATES DO
    asLookupKeys[nIterState] := '';
    abStateError[nIterState] := FALSE;
END_FOR

// Transition key is simple
asLookupKeys[0] := sTransitionKey;

// The other keys might be at different points in the astPositionState array.
// Try all of the posibilities, set error if we end up overwriting something.

// Outer loop: index of each motor at this position state
FOR nIterMotor := 1 TO MotionConstants.MAX_STATE_MOTORS DO
    // Inner loop: index of each position state for this motor
    FOR nIterState := 1 TO GeneralConstants.MAX_STATES DO
        sLoopNewKey := astPositionState[nIterMotor][nIterState].stPMPS.sPmpsState;
        IF sLoopNewKey <> '' THEN
            // We have a new key, start doing things
            sLoopPrevKey := asLookupKeys[nIterState];
            IF sLoopPrevKey = '' OR sLoopPrevKey = sLoopNewKey THEN
                // No key yet, or exactly the same key (redudant programmer)
                asLookupKeys[nIterState] := sLoopNewKey;
            ELSE
                // We already had a different key! Don't just override it, have an error!
                bError := TRUE;
                abStateError[nIterState] := TRUE;
            END_IF
        END_IF
    END_FOR
END_FOR

// Check for duplicated sPmpsState strings
FOR nIterState := 0 TO GeneralConstants.MAX_STATES DO
    FOR nIterState2 := 0 TO nIterState DO
        IF nIterState <> nIterState2 AND asLookupKeys[nIterState] = asLookupKeys[nIterState2] AND asLookupKeys[nIterState] <> '' THEN
            // Duplicated key, we need an error and a flag in both spots
            bError := TRUE;
            abStateError[nIterState] := TRUE;
            abStateError[nIterState2] := TRUE;
        END_IF
    END_FOR
END_FOR

// Clear the erroneous states so they won't be used as lookups
IF bError THEN
    FOR nIterState := 0 TO GeneralConstants.MAX_STATES DO
        IF abStateError[nIterState] THEN
            asLookupKeys[nIterState] := '';
        END_IF
    END_FOR
END_IF

// Copy the keys into the db state params
FOR nIterState := 0 TO GeneralConstants.MAX_STATES DO
    astDbStateParams[nIterState].sPmpsState := asLookupKeys[nIterState];
END_FOR

// Check if the keys changed from prev cycle
bNewKeys := FALSE;
FOR nIterState := 0 TO GeneralConstants.MAX_STATES DO
    IF asLookupKeys[nIterState] <> asPrevLookupKeys[nIterState] THEN
        bNewKeys := TRUE;
        EXIT;
    END_IF
END_FOR

// Save prev keys for next cycle
asPrevLookupKeys := asLookupKeys;
END_ACTION

END_FUNCTION_BLOCK

// ---- Tests/FB_MotionVirtualFrame_Test.TcPOU

FUNCTION_BLOCK FB_MotionVirtualFrame_Test EXTENDS TcUnit.FB_TestSuite
VAR
    nTestIDAssigner : INT;
    nTestID : INT := 1;
    tonTimeout : TON;
    tonStart : TON;

    stMotionStageRx : ST_MotionStage;
    stMotionStageRy : ST_MotionStage;
    stMotionStageRz : ST_MotionStage;

    stMotionStageVx : ST_MotionStage;
    stMotionStageVy : ST_MotionStage;
    stMotionStageVz : ST_MotionStage;

    fbMotionStageRx : FB_MotionStage;
    fbMotionStageRy : FB_MotionStage;
    fbMotionStageRz : FB_MotionStage;

    fbMotionStageVx : FB_MotionStage;
    fbMotionStageVy : FB_MotionStage;
    fbMotionStageVz : FB_MotionStage;

    nPositionCountsVx AT %Q* : UDINT;
    nPositionCountsVy AT %Q* : UDINT;
    nPositionCountsVz AT %Q* : UDINT;

    fbMotorTestSuite : FB_MotorTestSuite;
    fbMotionStageSetAndMoveHelper : FB_MotionStageSetAndMoveHelper;
    fbMotionStageSetHelperRx : FB_MotionStageSetHelper;
    fbMotionStageSetHelperRy : FB_MotionStageSetHelper;
    fbMotionStageSetHelperRz : FB_MotionStageSetHelper;
    fbMotionStageSetHelperVx : FB_MotionStageSetHelper;
    fbMotionStageSetHelperVy : FB_MotionStageSetHelper;
    fbMotionStageSetHelperVz : FB_MotionStageSetHelper;
    fbMotionVirtualFrame : FB_MotionVirtualFrame;
END_VAR


nTestIDAssigner := 0;

tonStart(IN := TRUE, PT := T#1s);

TestEnabled000045XYZMoveVxExpectNoErrorsCorrectPosVelAcc();

TestEnabled000090XYZMoveVxExpectNoErrorsCorrectPosVelAcc();

TestEnabled009090XYZMoveVxExpectNoErrorsCorrectPosVelAcc();

TestEnabled909090XYZMoveVxExpectNoErrorsCorrectPosVelAcc();

TestEnabledN22N21P4XYZMoveVxVyVzExpectNoErrorsCorrectPosVelAcc();

TestEnabledN22N21P4XYZMoveVyExpectNoErrorsCorrectPosVelAcc();

ACTION AssertNoErrors:

AssertFalse(
    Condition := tonTimeout.Q,
    Message := 'Timeout timer ended the test because it took longer than expected.'
);

AssertFalse(
    Condition := stMotionStageRx.bError,
    Message := 'Rx axis error detected when it should not have an error.'
);

AssertFalse(
    Condition := stMotionStageRy.bError,
    Message := 'Ry axis error detected when it should not have an error.'
);

AssertFalse(
    Condition := stMotionStageRz.bError,
    Message := 'Rz axis error detected when it should not have an error.'
);

AssertFalse(
    Condition := stMotionStageVx.bError,
    Message := 'Vx axis error detected when it should not have an error.'
);

AssertFalse(
    Condition := stMotionStageVy.bError,
    Message := 'Vy axis error detected when it should not have an error.'
);

AssertFalse(
    Condition := stMotionStageVz.bError,
    Message := 'Vz axis error detected when it should not have an error.'
);
END_ACTION


METHOD PRIVATE AssertPosVelAccCorrect
VAR_INPUT
    fDelta : LREAL;

    fRxPosExpected : LREAL;
    fRyPosExpected : LREAL;
    fRzPosExpected : LREAL;
    fVxPosExpected : LREAL;
    fVyPosExpected : LREAL;
    fVzPosExpected : LREAL;

    fRxVelExpected : LREAL;
    fRyVelExpected : LREAL;
    fRzVelExpected : LREAL;
    fVxVelExpected : LREAL;
    fVyVelExpected : LREAL;
    fVzVelExpected : LREAL;

    fRxAccExpected : LREAL;
    fRyAccExpected : LREAL;
    fRzAccExpected : LREAL;
    fVxAccExpected : LREAL;
    fVyAccExpected : LREAL;
    fVzAccExpected : LREAL;
END_VAR

// Position
AssertEquals_LREAL(
    Expected := fRxPosExpected,
    Actual := stMotionStageRx.Axis.NcToPlc.ActPos,
    Delta := fDelta,
    Message := 'Rx did not end at expected position.'
);

AssertEquals_LREAL(
    Expected := fRyPosExpected,
    Actual := stMotionStageRy.Axis.NcToPlc.ActPos,
    Delta := fDelta,
    Message := 'Ry did not end at expected position.'
);

AssertEquals_LREAL(
    Expected := fRzPosExpected,
    Actual := stMotionStageRz.Axis.NcToPlc.ActPos,
    Delta := fDelta,
    Message := 'Rz did not end at expected position.'
);

AssertEquals_LREAL(
    Expected := fVxPosExpected,
    Actual := stMotionStageVx.Axis.NcToPlc.ActPos,
    Delta := fDelta,
    Message := 'Vx did not end at expected position.'
);

AssertEquals_LREAL(
    Expected := fVyPosExpected,
    Actual := stMotionStageVy.Axis.NcToPlc.ActPos,
    Delta := fDelta,
    Message := 'Vy did not end at expected position.'
);

AssertEquals_LREAL(
    Expected := fVzPosExpected,
    Actual := stMotionStageVz.Axis.NcToPlc.ActPos,
    Delta := fDelta,
    Message := 'Vz did not end at expected position.'
);

// Velocity
AssertEquals_LREAL(
    Expected := fRxVelExpected,
    Actual := stMotionStageRx.fVelocity,
    Delta := fDelta,
    Message := 'Rx did not use the expected velocity.'
);

AssertEquals_LREAL(
    Expected := fRyVelExpected,
    Actual := stMotionStageRy.fVelocity,
    Delta := fDelta,
    Message := 'Ry did not use the expected velocity.'
);

AssertEquals_LREAL(
    Expected := fRzVelExpected,
    Actual := stMotionStageRz.fVelocity,
    Delta := fDelta,
    Message := 'Rz did not use the expected velocity.'
);

AssertEquals_LREAL(
    Expected := fVxVelExpected,
    Actual := stMotionStageVx.fVelocity,
    Delta := fDelta,
    Message := 'Vx did not use the expected velocity.'
);

AssertEquals_LREAL(
    Expected := fVyVelExpected,
    Actual := stMotionStageVy.fVelocity,
    Delta := fDelta,
    Message := 'Vy did not use the expected velocity.'
);

AssertEquals_LREAL(
    Expected := fVzVelExpected,
    Actual := stMotionStageVz.fVelocity,
    Delta := fDelta,
    Message := 'Vz did not use the expected velocity.'
);

// Acceleration
AssertEquals_LREAL(
    Expected := fRxAccExpected,
    Actual := stMotionStageRx.fAcceleration,
    Delta := fDelta,
    Message := 'Rx did not use the expected acceleration.'
);

AssertEquals_LREAL(
    Expected := fRyAccExpected,
    Actual := stMotionStageRy.fAcceleration,
    Delta := fDelta,
    Message := 'Ry did not use the expected acceleration.'
);

AssertEquals_LREAL(
    Expected := fRzAccExpected,
    Actual := stMotionStageRz.fAcceleration,
    Delta := fDelta,
    Message := 'Rz did not use the expected acceleration.'
);

AssertEquals_LREAL(
    Expected := fVxAccExpected,
    Actual := stMotionStageVx.fAcceleration,
    Delta := fDelta,
    Message := 'Vx did not use the expected acceleration.'
);

AssertEquals_LREAL(
    Expected := fVyAccExpected,
    Actual := stMotionStageVy.fAcceleration,
    Delta := fDelta,
    Message := 'Vy did not use the expected acceleration.'
);

AssertEquals_LREAL(
    Expected := fVzAccExpected,
    Actual := stMotionStageVz.fAcceleration,
    Delta := fDelta,
    Message := 'Vz did not use the expected acceleration.'
);
END_METHOD


METHOD PRIVATE InitMotors : BOOL

fbMotorTestSuite.SetEnables(stMotionStage := stMotionStageRx);
fbMotorTestSuite.SetEnables(stMotionStage := stMotionStageRy);
fbMotorTestSuite.SetEnables(stMotionStage := stMotionStageRz);
fbMotorTestSuite.SetEnables(stMotionStage := stMotionStageVx);
fbMotorTestSuite.SetEnables(stMotionStage := stMotionStageVy);
fbMotorTestSuite.SetEnables(stMotionStage := stMotionStageVz);

SetTar0();

fbMotionStageSetHelperRx(
    bExecute := TRUE,
    fStartPosition := 0.0,
    stMotionStage := stMotionStageRx,
    bResetDone => ,
    bSetDone =>
);

fbMotionStageSetHelperRy(
    bExecute := TRUE,
    fStartPosition := 0.0,
    stMotionStage := stMotionStageRy,
    bResetDone => ,
    bSetDone =>
);

fbMotionStageSetHelperRz(
    bExecute := TRUE,
    fStartPosition := 0.0,
    stMotionStage := stMotionStageRz,
    bResetDone => ,
    bSetDone =>
);

fbMotionStageSetHelperVx(
    bExecute := TRUE,
    fStartPosition := 0.0,
    stMotionStage := stMotionStageVx,
    bResetDone => ,
    bSetDone =>
);

fbMotionStageSetHelperVy(
    bExecute := TRUE,
    fStartPosition := 0.0,
    stMotionStage := stMotionStageVy,
    bResetDone => ,
    bSetDone =>
);

fbMotionStageSetHelperVz(
    bExecute := TRUE,
    fStartPosition := 0.0,
    stMotionStage := stMotionStageVz,
    bResetDone => ,
    bSetDone =>
);

IF fbMotionStageSetHelperRx.bSetDone AND
   fbMotionStageSetHelperRy.bSetDone AND
   fbMotionStageSetHelperRz.bSetDone AND
   fbMotionStageSetHelperVx.bSetDone AND
   fbMotionStageSetHelperVy.bSetDone AND
   fbMotionStageSetHelperVz.bSetDone THEN

    fbMotionStageSetHelperRx(
        bExecute := FALSE,
        fStartPosition := 0.0,
        stMotionStage := stMotionStageRx,
        bResetDone => ,
        bSetDone =>
    );

    fbMotionStageSetHelperRy(
        bExecute := FALSE,
        fStartPosition := 0.0,
        stMotionStage := stMotionStageRy,
        bResetDone => ,
        bSetDone =>
    );

    fbMotionStageSetHelperRz(
        bExecute := FALSE,
        fStartPosition := 0.0,
        stMotionStage := stMotionStageRz,
        bResetDone => ,
        bSetDone =>
    );

    fbMotionStageSetHelperVx(
        bExecute := FALSE,
        fStartPosition := 0.0,
        stMotionStage := stMotionStageVx,
        bResetDone => ,
        bSetDone =>
    );

    fbMotionStageSetHelperVy(
        bExecute := FALSE,
        fStartPosition := 0.0,
        stMotionStage := stMotionStageVy,
        bResetDone => ,
        bSetDone =>
    );

    fbMotionStageSetHelperVz(
        bExecute := FALSE,
        fStartPosition := 0.0,
        stMotionStage := stMotionStageVz,
        bResetDone => ,
        bSetDone =>
    );

    stMotionStageRx.nEnableMode := E_StageEnableMode.ALWAYS;
    stMotionStageRy.nEnableMode := E_StageEnableMode.ALWAYS;
    stMotionStageRz.nEnableMode := E_StageEnableMode.ALWAYS;
    stMotionStageVx.nEnableMode := E_StageEnableMode.ALWAYS;
    stMotionStageVy.nEnableMode := E_StageEnableMode.ALWAYS;
    stMotionStageVz.nEnableMode := E_StageEnableMode.ALWAYS;

    IF stMotionStageRx.bAllEnable AND
        stMotionStageRy.bAllEnable AND
        stMotionStageRz.bAllEnable AND
        stMotionStageVx.bAllEnable AND
        stMotionStageVy.bAllEnable AND
        stMotionStageVz.bAllEnable THEN

        InitMotors := TRUE;
    END_IF
END_IF
END_METHOD


METHOD PRIVATE SetTar0

stMotionStageVx.fPosition := 0.0;
stMotionStageVx.fVelocity := 0.0;
stMotionStageVx.fAcceleration := 0.0;

stMotionStageVy.fPosition := 0.0;
stMotionStageVy.fVelocity := 0.0;
stMotionStageVy.fAcceleration := 0.0;

stMotionStageVz.fPosition := 0.0;
stMotionStageVz.fVelocity := 0.0;
stMotionStageVz.fAcceleration := 0.0;

stMotionStageRx.fPosition := 0.0;
stMotionStageRx.fVelocity := 0.0;
stMotionStageRx.fAcceleration := 0.0;

stMotionStageRy.fPosition := 0.0;
stMotionStageRy.fVelocity := 0.0;
stMotionStageRy.fAcceleration := 0.0;

stMotionStageRz.fPosition := 0.0;
stMotionStageRz.fVelocity := 0.0;
stMotionStageRz.fAcceleration := 0.0;
END_METHOD


METHOD PRIVATE TestEnabled000045XYZMoveVxExpectNoErrorsCorrectPosVelAcc
VAR_INST
    bInit : BOOL;
    bComplete : BOOL;
    bBusyReached : BOOL;
    rtMoveCmdOnce : R_TRIG;
    fDelta : LREAL := 1e-9;
END_VAR

TEST('TestEnabled000045XYZMoveVxExpectNoErrorsCorrectPosVelAcc');

nTestIDAssigner := nTestIDAssigner + 1;

IF nTestID <> nTestIDAssigner OR NOT tonStart.Q THEN
    RETURN;
END_IF

tonTimeout(IN := TRUE, PT := T#3s);

IF NOT bInit THEN
    bInit := InitMotors();
END_IF

IF bInit THEN
    stMotionStageVx.fPosition := 15.0;
    stMotionStageVx.fVelocity := stMotionStageVx.fPosition * 2.0 / 3.0;
    stMotionStageVx.fAcceleration := stMotionStageVx.fVelocity * 5.0;
    rtMoveCmdOnce(CLK := TRUE);
    stMotionStageVx.bMoveCmd := rtMoveCmdOnce.Q;
END_IF

fbMotionVirtualFrame(
    stMotionStageRx := stMotionStageRx,
    stMotionStageRy := stMotionStageRy,
    stMotionStageRz := stMotionStageRz,
    stMotionStageVx := stMotionStageVx,
    stMotionStageVy := stMotionStageVy,
    stMotionStageVz := stMotionStageVz,
    bEnable := TRUE,
    fAlphaDegrees := 0.0,
    fBetaDegrees := 0.0,
    fGammaDegrees := 45.0,
    sOrder := 'XYZ',
    bBaseToNew := TRUE,
    fbVirtActPositionVec3 => ,
    fbVirtActVelocityVec3 => ,
    fbVirtActAcceleraVec3 =>
);

IF stMotionStageVx.bBusy THEN
    bBusyReached := TRUE;
END_IF

IF bBusyReached AND NOT stMotionStageVx.bBusy THEN
    bComplete := TRUE;
END_IF

IF (bComplete AND
    NOT stMotionStageVx.bBusy AND
    NOT stMotionStageVy.bBusy AND
    NOT stMotionStageVz.bBusy AND
    NOT stMotionStageRx.bBusy AND
    NOT stMotionStageRy.bBusy AND
    NOT stMotionStageRz.bBusy)
    OR tonTimeout.Q THEN

    AssertNoErrors();

    AssertPosVelAccCorrect(
        fDelta := fDelta,
        fRxPosExpected := stMotionStageVx.fPosition * SQRT(2.0) / 2.0,
        fRyPosExpected := stMotionStageVx.fPosition * SQRT(2.0) / 2.0,
        fRzPosExpected := 0.0,
        fVxPosExpected := stMotionStageVx.fPosition,
        fVyPosExpected := 0.0,
        fVzPosExpected := 0.0,
        fRxVelExpected := stMotionStageVx.fVelocity * SQRT(2.0) / 2.0,
        fRyVelExpected := stMotionStageVx.fVelocity * SQRT(2.0) / 2.0,
        fRzVelExpected := 0.0,
        fVxVelExpected := stMotionStageVx.fVelocity,
        fVyVelExpected := 0.0,
        fVzVelExpected := 0.0,
        fRxAccExpected := stMotionStageVx.fAcceleration * SQRT(2.0) / 2.0,
        fRyAccExpected := stMotionStageVx.fAcceleration * SQRT(2.0) / 2.0,
        fRzAccExpected := 0.0,
        fVxAccExpected := stMotionStageVx.fAcceleration,
        fVyAccExpected := 0.0,
        fVzAccExpected := 0.0
    );

    TEST_FINISHED();

    tonTimeout(IN := FALSE);

    nTestID := nTestID + 1;
END_IF

fbMotionStageRx(stMotionStage := stMotionStageRx);
fbMotionStageRy(stMotionStage := stMotionStageRy);
fbMotionStageRz(stMotionStage := stMotionStageRz);

fbMotionStageVx(stMotionStage := stMotionStageVx);
fbMotionStageVy(stMotionStage := stMotionStageVy);
fbMotionStageVz(stMotionStage := stMotionStageVz);

nPositionCountsVx := LREAL_TO_UDINT((fbMotionVirtualFrame.fbVirtActPositionVec3.x + 100.0) * 1e6);
nPositionCountsVy := LREAL_TO_UDINT((fbMotionVirtualFrame.fbVirtActPositionVec3.y + 100.0) * 1e6);
nPositionCountsVz := LREAL_TO_UDINT((fbMotionVirtualFrame.fbVirtActPositionVec3.z + 100.0) * 1e6);
END_METHOD


METHOD PRIVATE TestEnabled000090XYZMoveVxExpectNoErrorsCorrectPosVelAcc
VAR_INST
    bInit : BOOL;
    bComplete : BOOL;
    bBusyReached : BOOL;
    rtMoveCmdOnce : R_TRIG;
    fDelta : LREAL := 1e-9;
END_VAR

TEST('TestEnabled000090XYZMoveVxExpectNoErrorsCorrectPosVelAcc');

nTestIDAssigner := nTestIDAssigner + 1;

IF nTestID <> nTestIDAssigner OR NOT tonStart.Q THEN
    RETURN;
END_IF

tonTimeout(IN := TRUE, PT := T#3s);

IF NOT bInit THEN
    bInit := InitMotors();
END_IF

IF bInit THEN
    stMotionStageVx.fPosition := 20.0;
    stMotionStageVx.fVelocity := stMotionStageVx.fPosition * 2.0 / 3.0;
    stMotionStageVx.fAcceleration := stMotionStageVx.fVelocity * 5.0;
    rtMoveCmdOnce(CLK := TRUE);
    stMotionStageVx.bMoveCmd := rtMoveCmdOnce.Q;
END_IF

fbMotionVirtualFrame(
    stMotionStageRx := stMotionStageRx,
    stMotionStageRy := stMotionStageRy,
    stMotionStageRz := stMotionStageRz,
    stMotionStageVx := stMotionStageVx,
    stMotionStageVy := stMotionStageVy,
    stMotionStageVz := stMotionStageVz,
    bEnable := TRUE,
    fAlphaDegrees := 0.0,
    fBetaDegrees := 0.0,
    fGammaDegrees := 90.0,
    sOrder := 'XYZ',
    bBaseToNew := TRUE,
    fbVirtActPositionVec3 => ,
    fbVirtActVelocityVec3 => ,
    fbVirtActAcceleraVec3 =>
);

IF stMotionStageVx.bBusy THEN
    bBusyReached := TRUE;
END_IF

IF bBusyReached AND NOT stMotionStageVx.bBusy THEN
    bComplete := TRUE;
END_IF

IF (bComplete AND
    NOT stMotionStageVx.bBusy AND
    NOT stMotionStageVy.bBusy AND
    NOT stMotionStageVz.bBusy AND
    NOT stMotionStageRx.bBusy AND
    NOT stMotionStageRy.bBusy AND
    NOT stMotionStageRz.bBusy)
    OR tonTimeout.Q THEN

    AssertNoErrors();

    AssertPosVelAccCorrect(
        fDelta := fDelta,
        fRxPosExpected := 0.0,
        fRyPosExpected := stMotionStageVx.fPosition,
        fRzPosExpected := 0.0,
        fVxPosExpected := stMotionStageVx.fPosition,
        fVyPosExpected := 0.0,
        fVzPosExpected := 0.0,
        fRxVelExpected := 0.0,
        fRyVelExpected := stMotionStageVx.fVelocity,
        fRzVelExpected := 0.0,
        fVxVelExpected := stMotionStageVx.fVelocity,
        fVyVelExpected := 0.0,
        fVzVelExpected := 0.0,
        fRxAccExpected := 0.0,
        fRyAccExpected := stMotionStageVx.fAcceleration,
        fRzAccExpected := 0.0,
        fVxAccExpected := stMotionStageVx.fAcceleration,
        fVyAccExpected := 0.0,
        fVzAccExpected := 0.0
    );

    TEST_FINISHED();

    tonTimeout(IN := FALSE);

    nTestID := nTestID + 1;
END_IF

fbMotionStageRx(stMotionStage := stMotionStageRx);
fbMotionStageRy(stMotionStage := stMotionStageRy);
fbMotionStageRz(stMotionStage := stMotionStageRz);

fbMotionStageVx(stMotionStage := stMotionStageVx);
fbMotionStageVy(stMotionStage := stMotionStageVy);
fbMotionStageVz(stMotionStage := stMotionStageVz);

nPositionCountsVx := LREAL_TO_UDINT((fbMotionVirtualFrame.fbVirtActPositionVec3.x + 100.0) * 1e6);
nPositionCountsVy := LREAL_TO_UDINT((fbMotionVirtualFrame.fbVirtActPositionVec3.y + 100.0) * 1e6);
nPositionCountsVz := LREAL_TO_UDINT((fbMotionVirtualFrame.fbVirtActPositionVec3.z + 100.0) * 1e6);
END_METHOD


METHOD PRIVATE TestEnabled009090XYZMoveVxExpectNoErrorsCorrectPosVelAcc
VAR_INST
    bInit : BOOL;
    bComplete : BOOL;
    bBusyReached : BOOL;
    rtMoveCmdOnce : R_TRIG;
    fDelta : LREAL := 1e-9;
END_VAR

TEST('TestEnabled009090XYZMoveVxExpectNoErrorsCorrectPosVelAcc');

nTestIDAssigner := nTestIDAssigner + 1;

IF nTestID <> nTestIDAssigner OR NOT tonStart.Q THEN
    RETURN;
END_IF

tonTimeout(IN := TRUE, PT := T#3s);

IF NOT bInit THEN
    bInit := InitMotors();
END_IF

IF bInit THEN
    stMotionStageVx.fPosition := 25.0;
    stMotionStageVx.fVelocity := stMotionStageVx.fPosition * 2.0 / 3.0;
    stMotionStageVx.fAcceleration := stMotionStageVx.fVelocity * 5.0;
    rtMoveCmdOnce(CLK := TRUE);
    stMotionStageVx.bMoveCmd := rtMoveCmdOnce.Q;
END_IF

fbMotionVirtualFrame(
    stMotionStageRx := stMotionStageRx,
    stMotionStageRy := stMotionStageRy,
    stMotionStageRz := stMotionStageRz,
    stMotionStageVx := stMotionStageVx,
    stMotionStageVy := stMotionStageVy,
    stMotionStageVz := stMotionStageVz,
    bEnable := TRUE,
    fAlphaDegrees := 0.0,
    fBetaDegrees := 90.0,
    fGammaDegrees := 90.0,
    sOrder := 'XYZ',
    bBaseToNew := TRUE,
    fbVirtActPositionVec3 => ,
    fbVirtActVelocityVec3 => ,
    fbVirtActAcceleraVec3 =>
);

IF stMotionStageVx.bBusy THEN
    bBusyReached := TRUE;
END_IF

IF bBusyReached AND NOT stMotionStageVx.bBusy THEN
    bComplete := TRUE;
END_IF

IF (bComplete AND
    NOT stMotionStageVx.bBusy AND
    NOT stMotionStageVy.bBusy AND
    NOT stMotionStageVz.bBusy AND
    NOT stMotionStageRx.bBusy AND
    NOT stMotionStageRy.bBusy AND
    NOT stMotionStageRz.bBusy)
    OR tonTimeout.Q THEN

    AssertNoErrors();

    AssertPosVelAccCorrect(
        fDelta := fDelta,
        fRxPosExpected := 0.0,
        fRyPosExpected := stMotionStageVx.fPosition,
        fRzPosExpected := 0.0,
        fVxPosExpected := stMotionStageVx.fPosition,
        fVyPosExpected := 0.0,
        fVzPosExpected := 0.0,
        fRxVelExpected := 0.0,
        fRyVelExpected := stMotionStageVx.fVelocity,
        fRzVelExpected := 0.0,
        fVxVelExpected := stMotionStageVx.fVelocity,
        fVyVelExpected := 0.0,
        fVzVelExpected := 0.0,
        fRxAccExpected := 0.0,
        fRyAccExpected := stMotionStageVx.fAcceleration,
        fRzAccExpected := 0.0,
        fVxAccExpected := stMotionStageVx.fAcceleration,
        fVyAccExpected := 0.0,
        fVzAccExpected := 0.0
    );

    TEST_FINISHED();

    tonTimeout(IN := FALSE);

    nTestID := nTestID + 1;
END_IF

fbMotionStageRx(stMotionStage := stMotionStageRx);
fbMotionStageRy(stMotionStage := stMotionStageRy);
fbMotionStageRz(stMotionStage := stMotionStageRz);

fbMotionStageVx(stMotionStage := stMotionStageVx);
fbMotionStageVy(stMotionStage := stMotionStageVy);
fbMotionStageVz(stMotionStage := stMotionStageVz);

nPositionCountsVx := LREAL_TO_UDINT((fbMotionVirtualFrame.fbVirtActPositionVec3.x + 100.0) * 1e6);
nPositionCountsVy := LREAL_TO_UDINT((fbMotionVirtualFrame.fbVirtActPositionVec3.y + 100.0) * 1e6);
nPositionCountsVz := LREAL_TO_UDINT((fbMotionVirtualFrame.fbVirtActPositionVec3.z + 100.0) * 1e6);
END_METHOD


METHOD PRIVATE TestEnabled909090XYZMoveVxExpectNoErrorsCorrectPosVelAcc
VAR_INST
    bInit : BOOL;
    bComplete : BOOL;
    bBusyReached : BOOL;
    rtMoveCmdOnce : R_TRIG;
    fDelta : LREAL := 1e-9;
END_VAR

TEST('TestEnabled909090XYZMoveVxExpectNoErrorsCorrectPosVelAcc');

nTestIDAssigner := nTestIDAssigner + 1;

IF nTestID <> nTestIDAssigner OR NOT tonStart.Q THEN
    RETURN;
END_IF

tonTimeout(IN := TRUE, PT := T#3s);

IF NOT bInit THEN
    bInit := InitMotors();
END_IF

IF bInit THEN
    stMotionStageVx.fPosition := 35.0;
    stMotionStageVx.fVelocity := stMotionStageVx.fPosition * 2.0 / 3.0;
    stMotionStageVx.fAcceleration := stMotionStageVx.fVelocity * 5.0;
    rtMoveCmdOnce(CLK := TRUE);
    stMotionStageVx.bMoveCmd := rtMoveCmdOnce.Q;
END_IF

fbMotionVirtualFrame(
    stMotionStageRx := stMotionStageRx,
    stMotionStageRy := stMotionStageRy,
    stMotionStageRz := stMotionStageRz,
    stMotionStageVx := stMotionStageVx,
    stMotionStageVy := stMotionStageVy,
    stMotionStageVz := stMotionStageVz,
    bEnable := TRUE,
    fAlphaDegrees := 90.0,
    fBetaDegrees := 90.0,
    fGammaDegrees := 90.0,
    sOrder := 'XYZ',
    bBaseToNew := TRUE,
    fbVirtActPositionVec3 => ,
    fbVirtActVelocityVec3 => ,
    fbVirtActAcceleraVec3 =>
);

IF stMotionStageVx.bBusy THEN
    bBusyReached := TRUE;
END_IF

IF bBusyReached AND NOT stMotionStageVx.bBusy THEN
    bComplete := TRUE;
END_IF

IF (bComplete AND
    NOT stMotionStageVx.bBusy AND
    NOT stMotionStageVy.bBusy AND
    NOT stMotionStageVz.bBusy AND
    NOT stMotionStageRx.bBusy AND
    NOT stMotionStageRy.bBusy AND
    NOT stMotionStageRz.bBusy)
    OR tonTimeout.Q THEN

    AssertNoErrors();

    AssertPosVelAccCorrect(
        fDelta := fDelta,
        fRxPosExpected := 0.0,
        fRyPosExpected := 0.0,
        fRzPosExpected := stMotionStageVx.fPosition,
        fVxPosExpected := stMotionStageVx.fPosition,
        fVyPosExpected := 0.0,
        fVzPosExpected := 0.0,
        fRxVelExpected := 0.0,
        fRyVelExpected := 0.0,
        fRzVelExpected := stMotionStageVx.fVelocity,
        fVxVelExpected := stMotionStageVx.fVelocity,
        fVyVelExpected := 0.0,
        fVzVelExpected := 0.0,
        fRxAccExpected := 0.0,
        fRyAccExpected := 0.0,
        fRzAccExpected := stMotionStageVx.fAcceleration,
        fVxAccExpected := stMotionStageVx.fAcceleration,
        fVyAccExpected := 0.0,
        fVzAccExpected := 0.0
    );

    TEST_FINISHED();

    tonTimeout(IN := FALSE);

    nTestID := nTestID + 1;
END_IF

fbMotionStageRx(stMotionStage := stMotionStageRx);
fbMotionStageRy(stMotionStage := stMotionStageRy);
fbMotionStageRz(stMotionStage := stMotionStageRz);

fbMotionStageVx(stMotionStage := stMotionStageVx);
fbMotionStageVy(stMotionStage := stMotionStageVy);
fbMotionStageVz(stMotionStage := stMotionStageVz);

nPositionCountsVx := LREAL_TO_UDINT((fbMotionVirtualFrame.fbVirtActPositionVec3.x + 100.0) * 1e6);
nPositionCountsVy := LREAL_TO_UDINT((fbMotionVirtualFrame.fbVirtActPositionVec3.y + 100.0) * 1e6);
nPositionCountsVz := LREAL_TO_UDINT((fbMotionVirtualFrame.fbVirtActPositionVec3.z + 100.0) * 1e6);
END_METHOD


METHOD PRIVATE TestEnabledN22N21P4XYZMoveVxVyVzExpectNoErrorsCorrectPosVelAcc
VAR_INST
    bInit : BOOL;
    bComplete : BOOL;
    bBusyReached : BOOL;
    rtMoveCmdOnce : R_TRIG;
    fDelta : LREAL := 1e-9;
END_VAR

TEST('TestEnabledN22N21P4XYZMoveVxVyVzExpectNoErrorsCorrectPosVelAcc');

nTestIDAssigner := nTestIDAssigner + 1;

IF nTestID <> nTestIDAssigner OR NOT tonStart.Q THEN
    RETURN;
END_IF

tonTimeout(IN := TRUE, PT := T#3s);

IF NOT bInit THEN
    bInit := InitMotors();
END_IF

IF bInit THEN
    rtMoveCmdOnce(CLK := TRUE);

    stMotionStageVx.fPosition := 15.0;
    stMotionStageVx.fVelocity := stMotionStageVx.fPosition * 2.0 / 3.0;
    stMotionStageVx.fAcceleration := stMotionStageVx.fVelocity * 5.0;
    stMotionStageVx.bMoveCmd := rtMoveCmdOnce.Q;

    stMotionStageVy.fPosition := -30.0;
    stMotionStageVy.fVelocity := ABS(stMotionStageVy.fPosition * 2.0 / 3.0);
    stMotionStageVy.fAcceleration := ABS(stMotionStageVy.fVelocity * 5.0);
    stMotionStageVy.bMoveCmd := rtMoveCmdOnce.Q;

    stMotionStageVz.fPosition := 45.0;
    stMotionStageVz.fVelocity := stMotionStageVz.fPosition * 2.0 / 3.0;
    stMotionStageVz.fAcceleration := stMotionStageVz.fVelocity * 5.0;
    stMotionStageVz.bMoveCmd := rtMoveCmdOnce.Q;
END_IF

fbMotionVirtualFrame(
    stMotionStageRx := stMotionStageRx,
    stMotionStageRy := stMotionStageRy,
    stMotionStageRz := stMotionStageRz,
    stMotionStageVx := stMotionStageVx,
    stMotionStageVy := stMotionStageVy,
    stMotionStageVz := stMotionStageVz,
    bEnable := TRUE,
    fAlphaDegrees := -22.21,
    fBetaDegrees := -20.7,
    fGammaDegrees := 3.793,
    sOrder := 'XYZ',
    bBaseToNew := FALSE,
    fbVirtActPositionVec3 => ,
    fbVirtActVelocityVec3 => ,
    fbVirtActAcceleraVec3 =>
);

IF stMotionStageVx.bBusy AND stMotionStageVy.bBusy AND stMotionStageVz.bBusy THEN
    bBusyReached := TRUE;
END_IF

IF bBusyReached AND NOT stMotionStageVx.bBusy AND NOT stMotionStageVy.bBusy AND NOT stMotionStageVz.bBusy THEN
    bComplete := TRUE;
END_IF

IF (bComplete AND
    NOT stMotionStageVx.bBusy AND
    NOT stMotionStageVy.bBusy AND
    NOT stMotionStageVz.bBusy AND
    NOT stMotionStageRx.bBusy AND
    NOT stMotionStageRy.bBusy AND
    NOT stMotionStageRz.bBusy)
    OR tonTimeout.Q THEN

    AssertNoErrors();

    AssertPosVelAccCorrect(
        fDelta := fDelta,
        fRxPosExpected := 21.732640182123049,
        fRyPosExpected := -46.323371856381527,
        fRzPosExpected := 23.061603816078627,
        fVxPosExpected := stMotionStageVx.fPosition,
        fVyPosExpected := stMotionStageVy.fPosition,
        fVzPosExpected := stMotionStageVz.fPosition,
        fRxVelExpected := 14.488426788082032,
        fRyVelExpected := 30.882247904254346,
        fRzVelExpected := 15.374402544052412,
        fVxVelExpected := stMotionStageVx.fVelocity,
        fVyVelExpected := stMotionStageVy.fVelocity,
        fVzVelExpected := stMotionStageVz.fVelocity,
        fRxAccExpected := 0.724421339404102 * 1e2,
        fRyAccExpected := 1.544112395212718 * 1e2,
        fRzAccExpected := 0.768720127202621 * 1e2,
        fVxAccExpected := stMotionStageVx.fAcceleration,
        fVyAccExpected := stMotionStageVy.fAcceleration,
        fVzAccExpected := stMotionStageVz.fAcceleration
    );

    TEST_FINISHED();

    tonTimeout(IN := FALSE);

    nTestID := nTestID + 1;
END_IF

fbMotionStageRx(stMotionStage := stMotionStageRx);
fbMotionStageRy(stMotionStage := stMotionStageRy);
fbMotionStageRz(stMotionStage := stMotionStageRz);

fbMotionStageVx(stMotionStage := stMotionStageVx);
fbMotionStageVy(stMotionStage := stMotionStageVy);
fbMotionStageVz(stMotionStage := stMotionStageVz);

nPositionCountsVx := LREAL_TO_UDINT((fbMotionVirtualFrame.fbVirtActPositionVec3.x + 100.0) * 1e6);
nPositionCountsVy := LREAL_TO_UDINT((fbMotionVirtualFrame.fbVirtActPositionVec3.y + 100.0) * 1e6);
nPositionCountsVz := LREAL_TO_UDINT((fbMotionVirtualFrame.fbVirtActPositionVec3.z + 100.0) * 1e6);
END_METHOD


METHOD PRIVATE TestEnabledN22N21P4XYZMoveVyExpectNoErrorsCorrectPosVelAcc
VAR_INST
    bInit : BOOL;
    bComplete : BOOL;
    bBusyReached : BOOL;
    rtMoveCmdOnce : R_TRIG;
    fDelta : LREAL := 1e-9;
END_VAR

TEST('TestEnabledN22N21P4XYZMoveVyExpectNoErrorsCorrectPosVelAcc');

nTestIDAssigner := nTestIDAssigner + 1;

IF nTestID <> nTestIDAssigner OR NOT tonStart.Q THEN
    RETURN;
END_IF

tonTimeout(IN := TRUE, PT := T#3s);

IF NOT bInit THEN
    bInit := InitMotors();
END_IF

IF bInit THEN
    stMotionStageVy.fPosition := 30.0;
    stMotionStageVy.fVelocity := stMotionStageVy.fPosition * 2.0 / 3.0;
    stMotionStageVy.fAcceleration := stMotionStageVy.fVelocity * 5.0;
    rtMoveCmdOnce(CLK := TRUE);
    stMotionStageVy.bMoveCmd := rtMoveCmdOnce.Q;
END_IF

fbMotionVirtualFrame(
    stMotionStageRx := stMotionStageRx,
    stMotionStageRy := stMotionStageRy,
    stMotionStageRz := stMotionStageRz,
    stMotionStageVx := stMotionStageVx,
    stMotionStageVy := stMotionStageVy,
    stMotionStageVz := stMotionStageVz,
    bEnable := TRUE,
    fAlphaDegrees := -22.21,
    fBetaDegrees := -20.7,
    fGammaDegrees := 3.793,
    sOrder := 'XYZ',
    bBaseToNew := FALSE,
    fbVirtActPositionVec3 => ,
    fbVirtActVelocityVec3 => ,
    fbVirtActAcceleraVec3 =>
);

IF stMotionStageVy.bBusy THEN
    bBusyReached := TRUE;
END_IF

IF bBusyReached AND NOT stMotionStageVy.bBusy THEN
    bComplete := TRUE;
END_IF

IF (bComplete AND
    NOT stMotionStageVx.bBusy AND
    NOT stMotionStageVy.bBusy AND
    NOT stMotionStageVz.bBusy AND
    NOT stMotionStageRx.bBusy AND
    NOT stMotionStageRy.bBusy AND
    NOT stMotionStageRz.bBusy)
    OR tonTimeout.Q THEN

    AssertNoErrors();

    AssertPosVelAccCorrect(
        fDelta := fDelta,
        fRxPosExpected := 5.836964390001455,
        fRyPosExpected := 27.448135465863341,
        fRzPosExpected := 10.608001987060069,
        fVxPosExpected := 0.0,
        fVyPosExpected := stMotionStageVy.fPosition,
        fVzPosExpected := 0.0,
        fRxVelExpected := 5.836964390001455 * 2.0 / 3.0,
        fRyVelExpected := 27.448135465863341 * 2.0 / 3.0,
        fRzVelExpected := 10.608001987060069 * 2.0 / 3.0,
        fVxVelExpected := 0.0,
        fVyVelExpected := stMotionStageVy.fVelocity,
        fVzVelExpected := 0.0,
        fRxAccExpected := 5.836964390001455 * 2.0 / 3.0 * 5.0,
        fRyAccExpected := 27.448135465863341 * 2.0 / 3.0 * 5.0,
        fRzAccExpected := 10.608001987060069 * 2.0 / 3.0 * 5.0,
        fVxAccExpected := 0.0,
        fVyAccExpected := stMotionStageVy.fAcceleration,
        fVzAccExpected := 0.0
    );

    TEST_FINISHED();

    tonTimeout(IN := FALSE);

    nTestID := nTestID + 1;
END_IF

fbMotionStageRx(stMotionStage := stMotionStageRx);
fbMotionStageRy(stMotionStage := stMotionStageRy);
fbMotionStageRz(stMotionStage := stMotionStageRz);

fbMotionStageVx(stMotionStage := stMotionStageVx);
fbMotionStageVy(stMotionStage := stMotionStageVy);
fbMotionStageVz(stMotionStage := stMotionStageVz);

nPositionCountsVx := LREAL_TO_UDINT((fbMotionVirtualFrame.fbVirtActPositionVec3.x + 100.0) * 1e6);
nPositionCountsVy := LREAL_TO_UDINT((fbMotionVirtualFrame.fbVirtActPositionVec3.y + 100.0) * 1e6);
nPositionCountsVz := LREAL_TO_UDINT((fbMotionVirtualFrame.fbVirtActPositionVec3.z + 100.0) * 1e6);
END_METHOD

END_FUNCTION_BLOCK

// ---- Tests/Helpers/FB_MotionStageSetAndMoveHelper.TcPOU
FUNCTION_BLOCK FB_MotionStageSetAndMoveHelper
VAR_INPUT
    // Begin on rising edge, stop on falling edge.
    bExecute: BOOL;
    // The position to set the motor to
    fStartPosition: LREAL;
    // The goal to move the motor towards
    fGoalPosition: LREAL;
    // The velocity to move at
    fVelocity: LREAL;
    // The allowable deviation from the goal position to be considered done moving.
    fDelta: LREAL;
END_VAR
VAR_IN_OUT
    stMotionStage: ST_MotionStage;
END_VAR
VAR_OUTPUT
    // Goes to TRUE once the motor has no errors and is deactivated.
    bResetDone: BOOL;
    // Goes to TRUE once the set position completes.
    bSetDone: BOOL;
    // Goes to TRUE once the motor begins moving.
    bMotionStarted: BOOL;
    // Goes to TRUE once the motor reaches its destination.
    bMoveDone: BOOL;
END_VAR
VAR
    rtExec: R_TRIG;
    mcSetPos: MC_SetPosition;
END_VAR

rtExec(CLK:=bExecute);

IF rtExec.Q THEN
    stMotionStage.bReset := TRUE;
    stMotionStage.bEnable := FALSE;
    stMotionStage.nEnableMode := E_StageEnableMode.NEVER;
    mcSetPos(
        Axis:=stMotionStage.Axis,
        Execute:=FALSE
    );
    bResetDone := FALSE;
    bSetDone := FALSE;
    bMotionStarted := FALSE;
    bMoveDone := FALSE;
END_IF

bResetDone := NOT stMotionStage.bError AND NOT stMotionStage.bBusy;
bMoveDone := stMotionStage.Axis.NcToPlc.ActPos <= fGoalPosition + fDelta AND
             stMotionStage.Axis.NcToPlc.ActPos >= fGoalPosition - fDelta;

IF NOT bSetDone THEN
    stMotionStage.bReset := TRUE;
    stMotionStage.bEnable := FALSE;
    IF stMotionStage.stAxisStatus.fActPosition <> fStartPosition THEN
        mcSetPos(
            Axis:=stMotionStage.Axis,
            Execute:=NOT mcSetPos.Execute,
            Position:=fStartPosition,
            Mode:=FALSE,
            Done=>
        );
    ELSE
        bSetDone := TRUE;
    END_IF
ELSE
    stMotionStage.bEnable := TRUE;
    IF NOT bMotionStarted AND NOT stMotionStage.Axis.Status.Disabled THEN
        stMotionStage.fPosition := fGoalPosition;
        stMotionStage.fVelocity := fVelocity;
        stMotionStage.bMoveCmd := TRUE;
        bMotionStarted := TRUE;
    END_IF
END_IF

IF bMoveDone THEN
    stMotionStage.bReset := TRUE;
END_IF


METHOD PUBLIC Reset
VAR_IN_OUT
    stMotionStage : ST_MotionStage;
END_VAR

rtExec(CLK:=FALSE);

stMotionStage.bReset := FALSE;
stMotionStage.bEnable := FALSE;
stMotionStage.nEnableMode := E_StageEnableMode.NEVER;
mcSetPos(
    Axis:=stMotionStage.Axis,
    Execute:=FALSE
);
bResetDone := FALSE;
bSetDone := FALSE;
bMotionStarted := FALSE;
bMoveDone := FALSE;
END_METHOD

END_FUNCTION_BLOCK

// ---- Tests/Helpers/FB_MotionStageSetHelper.TcPOU
FUNCTION_BLOCK FB_MotionStageSetHelper
VAR_INPUT
    // Begin on rising edge, stop on falling edge.
    bExecute: BOOL;
    // The position to set the motor to
    fStartPosition: LREAL;
END_VAR
VAR_IN_OUT
    stMotionStage: ST_MotionStage;
END_VAR
VAR_OUTPUT
    // Goes to TRUE once the motor has no errors and is deactivated.
    bResetDone: BOOL;
    // Goes to TRUE once the set position completes.
    bSetDone: BOOL;
END_VAR
VAR
    rtExec: R_TRIG;
    mcSetPos: MC_SetPosition;
    stSetPositionOptions : ST_SetPositionOptions;
END_VAR


rtExec(CLK:=bExecute);

IF rtExec.Q THEN
    stMotionStage.bReset := TRUE;
    stMotionStage.bEnable := FALSE;
    stMotionStage.nEnableMode := E_StageEnableMode.NEVER;
    mcSetPos(
        Axis:=stMotionStage.Axis,
        Execute:=FALSE
    );
    bResetDone := FALSE;
    bSetDone := FALSE;
END_IF

bResetDone := NOT stMotionStage.bError AND NOT stMotionStage.bBusy;

IF bResetDone THEN
    stMotionStage.bReset := FALSE;
END_IF

IF NOT bSetDone THEN
    stMotionStage.bEnable := FALSE;
    IF stMotionStage.Axis.NcToPlc.ActPos <> fStartPosition THEN
        stSetPositionOptions.ClearPositionLag := TRUE;
        mcSetPos(
            Axis:=stMotionStage.Axis,
            Execute:=NOT mcSetPos.Execute,
            Position:=fStartPosition,
            Mode:=FALSE,
            Options:=stSetPositionOptions,
            Done=>
        );
    ELSE
        bSetDone := TRUE;
    END_IF
END_IF

END_FUNCTION_BLOCK

// ---- POUs/Motion/FB_MotionVirtualFrame.TcPOU

FUNCTION_BLOCK FB_MotionVirtualFrame
(*
Takes 3 ST_MotionStages representing real axes that are orthogonal to each other and in a base frame of reference.
Takes 3 ST_MotionStages representing virtual axes that are orthogonal to each other and in a new frame of reference.
Computes the transformation from the base to the new frame of reference using 3 euler angles and a rotation order
as inputs. By default, the order and angles are interpreted as going from the base to the virtual frame. Can be
switched to go from virtual to base frame of reference.
If enabled, this function block will automatically handle commanding the real axes to move when the virtual axes
are commanded to move. If not enabled, the function block acts as a calculator, outputing the results of
calculating motions in a new frame of reference, but not changing any setpoints or commanding any moves.
*)
VAR_IN_OUT
    stMotionStageRx : ST_MotionStage; // Real X Axis in base frame of reference
    stMotionStageRy : ST_MotionStage; // Real Y Axis in base frame of reference
    stMotionStageRz : ST_MotionStage; // Real Z Axis in base frame of reference
    stMotionStageVx : ST_MotionStage; // Virtual X Axis in new frame of reference
    stMotionStageVy : ST_MotionStage; // Virtual Y Axis in new frame of reference
    stMotionStageVz : ST_MotionStage; // Virtual Z Axis in new frame of reference
END_VAR
VAR_INPUT
    (*TRUE to automatically overwrite real axis setpoints and command moves.
      FALSE to use this function only as a calculator.*)
    bEnable : BOOL;
    fAlphaDegrees : LREAL; // Angle of rotation about first axis.
    fBetaDegrees : LREAL; // Angle of rotation about second axis.
    fGammaDegrees : LREAL; // Angle of rotation about third axis.
    (*Rotation Order. E.g: XYZ to rotate alpha degrees around X axis, beta degrees around Y axis,
      and gamma degrees around Z axis. Valid rotation orders are:
      YZY, YXY, ZYZ, ZXZ, XYX, XZX, XYZ, YZX, ZXY, XZY, ZYX, YXZ.
      Default order for empty or invalid input is: ZYX.*)
    sOrder : STRING;
    (*FALSE to define inputs as rotating the frame of reference from the new frame to the base frame.
      TRUE to define the inputs as rotating the frame of reference from the base from to the new frame.*)
    bBaseToNew : BOOL := TRUE;
END_VAR
VAR_OUTPUT
    fbVirtActPositionVec3 : FB_Vec3;
    fbVirtActVelocityVec3 : FB_Vec3;
    fbVirtActAcceleraVec3 : FB_Vec3;

    fbRealTarPositionVec3 : FB_Vec3;
    fbRealTarVelocityVec3 : FB_Vec3;
    fbRealTarAcceleraVec3 : FB_Vec3;
END_VAR
VAR
    fAlphaRadians : LREAL;
    fBetaRadians : LREAL;
    fGammaRadians : LREAL;

    rtExecuteVx : R_TRIG;
    rtExecuteVy : R_TRIG;
    rtExecuteVz : R_TRIG;

    fbRealActPositionVec3 : FB_Vec3;
    fbRealActVelocityVec3 : FB_Vec3;
    fbRealActAcceleraVec3 : FB_Vec3;

    sOrderReversed : STRING;
    sLeft : STRING;
    sMid : STRING;
    sRight : STRING;

    fbVirtTarPositionVec3 : FB_Vec3;
    fbVirtTarVelocityVec3 : FB_Vec3;
    fbVirtTarAcceleraVec3 : FB_Vec3;
END_VAR


fAlphaRadians := DegToRad(fAlphaDegrees);
fBetaRadians := DegToRad(fBetaDegrees);
fGammaRadians := DegToRad(fGammaDegrees);

rtExecuteVx(CLK := stMotionStageVx.bBusy);
rtExecuteVy(CLK := stMotionStageVy.bBusy);
rtExecuteVz(CLK := stMotionStageVz.bBusy);

fbRealActPositionVec3.x := stMotionStageRx.Axis.NcToPlc.ActPos;
fbRealActPositionVec3.y := stMotionStageRy.Axis.NcToPlc.ActPos;
fbRealActPositionVec3.z := stMotionStageRz.Axis.NcToPlc.ActPos;

fbRealActVelocityVec3.x := stMotionStageRx.Axis.NcToPlc.ActVelo;
fbRealActVelocityVec3.y := stMotionStageRy.Axis.NcToPlc.ActVelo;
fbRealActVelocityVec3.z := stMotionStageRz.Axis.NcToPlc.ActVelo;

fbRealActAcceleraVec3.x := stMotionStageRx.Axis.NcToPlc.ActAcc;
fbRealActAcceleraVec3.y := stMotionStageRy.Axis.NcToPlc.ActAcc;
fbRealActAcceleraVec3.z := stMotionStageRz.Axis.NcToPlc.ActAcc;

sOrderReversed := ReverseOrder(sOrder);

IF bBaseToNew THEN
    RotatePosVelAccFrame(
        fbBaseFramePositionVec3 := fbRealActPositionVec3,
        fbBaseFrameVelocityVec3 := fbRealActVelocityVec3,
        fbBaseFrameAcceleraVec3 := fbRealActAcceleraVec3,
        fbNewFramePositionVec3 => fbVirtActPositionVec3,
        fbNewFrameVelocityVec3 => fbVirtActVelocityVec3,
        fbNewFrameAcceleraVec3 => fbVirtActAcceleraVec3,
        fAlphaRadians := fAlphaRadians,
        fBetaRadians := fBetaRadians,
        fGammaRadians := fGammaRadians,
        sOrder := sOrder
    );
ELSE
    RotatePosVelAccFrame(
        fbBaseFramePositionVec3 := fbRealActPositionVec3,
        fbBaseFrameVelocityVec3 := fbRealActVelocityVec3,
        fbBaseFrameAcceleraVec3 := fbRealActAcceleraVec3,
        fbNewFramePositionVec3 => fbVirtActPositionVec3,
        fbNewFrameVelocityVec3 => fbVirtActVelocityVec3,
        fbNewFrameAcceleraVec3 => fbVirtActAcceleraVec3,
        fAlphaRadians := -fGammaRadians,
        fBetaRadians := -fBetaRadians,
        fGammaRadians := -fAlphaRadians,
        sOrder := sOrderReversed
    );
END_IF

SetTargetPosVelAcc3D(
    stMotionStageX := stMotionStageVx,
    stMotionStageY := stMotionStageVy,
    stMotionStageZ := stMotionStageVz,
    fbActPosVec3 := fbVirtActPositionVec3,
    fbTarPosVec3 => fbVirtTarPositionVec3,
    fbTarVelVec3 => fbVirtTarVelocityVec3,
    fbTarAccVec3 => fbVirtTarAcceleraVec3
);

IF bBaseToNew THEN
    RotatePosVelAccFrame(
        fbBaseFramePositionVec3 := fbVirtTarPositionVec3,
        fbBaseFrameVelocityVec3 := fbVirtTarVelocityVec3,
        fbBaseFrameAcceleraVec3 := fbVirtTarAcceleraVec3,
        fbNewFramePositionVec3 => fbRealTarPositionVec3,
        fbNewFrameVelocityVec3 => fbRealTarVelocityVec3,
        fbNewFrameAcceleraVec3 => fbRealTarAcceleraVec3,
        fAlphaRadians := -fGammaRadians,
        fBetaRadians := -fBetaRadians,
        fGammaRadians := -fAlphaRadians,
        sOrder := sOrderReversed
    );
ELSE
    RotatePosVelAccFrame(
        fbBaseFramePositionVec3 := fbVirtTarPositionVec3,
        fbBaseFrameVelocityVec3 := fbVirtTarVelocityVec3,
        fbBaseFrameAcceleraVec3 := fbVirtTarAcceleraVec3,
        fbNewFramePositionVec3 => fbRealTarPositionVec3,
        fbNewFrameVelocityVec3 => fbRealTarVelocityVec3,
        fbNewFrameAcceleraVec3 => fbRealTarAcceleraVec3,
        fAlphaRadians := fAlphaRadians,
        fBetaRadians := fBetaRadians,
        fGammaRadians := fGammaRadians,
        sOrder := sOrder
    );
END_IF

IF bEnable THEN
    IF rtExecuteVx.Q OR rtExecuteVy.Q OR rtExecuteVz.Q THEN
        stMotionStageRx.fPosition := fbRealTarPositionVec3.x;
        stMotionStageRy.fPosition := fbRealTarPositionVec3.y;
        stMotionStageRz.fPosition := fbRealTarPositionVec3.z;

        stMotionStageRx.fVelocity := ABS(fbRealTarVelocityVec3.x);
        stMotionStageRy.fVelocity := ABS(fbRealTarVelocityVec3.y);
        stMotionStageRz.fVelocity := ABS(fbRealTarVelocityVec3.z);

        stMotionStageRx.fAcceleration := ABS(fbRealTarAcceleraVec3.x);
        stMotionStageRy.fAcceleration := ABS(fbRealTarAcceleraVec3.y);
        stMotionStageRz.fAcceleration := ABS(fbRealTarAcceleraVec3.z);

        stMotionStageRx.fDeceleration := ABS(fbRealTarAcceleraVec3.x);
        stMotionStageRy.fDeceleration := ABS(fbRealTarAcceleraVec3.y);
        stMotionStageRz.fDeceleration := ABS(fbRealTarAcceleraVec3.z);

        IF stMotionStageRx.fVelocity >= 0.001 THEN
            stMotionStageRx.bMoveCmd := TRUE;
        ELSIF ABS(stMotionStageRx.fPosition - stMotionStageRx.Axis.NcToPlc.ActPos) >
                stMotionStageRx.stAxisParameters.fTargetPosControlRange THEN
            stMotionStageRx.fVelocity := 0.001;
            stMotionStageRx.bMoveCmd := TRUE;
        END_IF

        IF stMotionStageRy.fVelocity >= 0.001 THEN
            stMotionStageRy.bMoveCmd := TRUE;
        ELSIF ABS(stMotionStageRy.fPosition - stMotionStageRy.Axis.NcToPlc.ActPos) >
                stMotionStageRy.stAxisParameters.fTargetPosControlRange THEN
            stMotionStageRy.fVelocity := 0.001;
            stMotionStageRy.bMoveCmd := TRUE;
        END_IF

        IF stMotionStageRz.fVelocity >= 0.001 THEN
            stMotionStageRz.bMoveCmd := TRUE;
        ELSIF ABS(stMotionStageRz.fPosition - stMotionStageRz.Axis.NcToPlc.ActPos) >
                stMotionStageRz.stAxisParameters.fTargetPosControlRange THEN
            stMotionStageRz.fVelocity := 0.001;
            stMotionStageRz.bMoveCmd := TRUE;
        END_IF
    END_IF

    IF stMotionStageRx.bError OR stMotionStageRy.bError OR stMotionStageRz.bError THEN
        stMotionStageVx.bError := TRUE;
        stMotionStageVy.bError := TRUE;
        stMotionStageVz.bError := TRUE;
        stMotionStageVx.sCustomErrorMessage := 'An error occured in one of the real axes. All virtual axes stopped.';
        stMotionStageVy.sCustomErrorMessage := 'An error occured in one of the real axes. All virtual axes stopped.';
        stMotionStageVz.sCustomErrorMessage := 'An error occured in one of the real axes. All virtual axes stopped.';
    END_IF
END_IF


METHOD PUBLIC DegToRad : LREAL
VAR_INPUT
    fDeg : LREAL;
END_VAR

DegToRad := fDeg  / 180.0 * lcls_twincat_math.GVL_Constants.PI;
END_METHOD

METHOD ReverseOrder : STRING
VAR_INPUT
    sOrder : STRING;
END_VAR

IF sOrder = '' THEN
    sOrder := 'ZYX';
END_IF
sLeft := LEFT(sOrder, 1);
sMid := MID(sOrder, 1, 2);
sRight := RIGHT(sOrder, 1);
ReverseOrder := CONCAT(sRight, CONCAT(sMid, sLeft));
END_METHOD


METHOD PUBLIC RotatePosVelAccFrame
VAR_INPUT
    fbBaseFramePositionVec3 : FB_Vec3;
    fbBaseFrameVelocityVec3 : FB_Vec3;
    fbBaseFrameAcceleraVec3 : FB_Vec3;

    fAlphaRadians : LREAL;
    fBetaRadians : LREAL;
    fGammaRadians : LREAL;
    sOrder : STRING;
END_VAR
VAR_OUTPUT
    fbNewFramePositionVec3 : FB_Vec3;
    fbNewFrameVelocityVec3 : FB_Vec3;
    fbNewFrameAcceleraVec3 : FB_Vec3;
END_VAR

fbNewFramePositionVec3 := F_EulerRotateVec3Frame(
    iVec3 := fbBaseFramePositionVec3,
    fAlphaRadians := fAlphaRadians,
    fBetaRadians := fBetaRadians,
    fGammaRadians := fGammaRadians,
    sOrder := sOrder
);

fbNewFrameVelocityVec3 := F_EulerRotateVec3Frame(
    iVec3 := fbBaseFrameVelocityVec3,
    fAlphaRadians := fAlphaRadians,
    fBetaRadians := fBetaRadians,
    fGammaRadians := fGammaRadians,
    sOrder := sOrder
);

fbNewFrameAcceleraVec3 := F_EulerRotateVec3Frame(
    iVec3 := fbBaseFrameAcceleraVec3,
    fAlphaRadians := fAlphaRadians,
    fBetaRadians := fBetaRadians,
    fGammaRadians := fGammaRadians,
    sOrder := sOrder
);
END_METHOD


METHOD PUBLIC SetTargetPosVelAcc1D
VAR_INPUT
    stMotionStage : ST_MotionStage;
    fActPos : LREAL;
END_VAR
VAR_OUTPUT
    fTarPos : LREAL;
    fTarVel : LREAL;
    fTarAcc : LREAL;
END_VAR

IF stMotionStage.bBusy THEN
    fTarPos := stMotionStage.fPosition;
    IF fTarPos >= fActPos THEN
        fTarVel := stMotionStage.fVelocity;
        fTarAcc := stMotionStage.fAcceleration;
    ELSE
        fTarVel := -stMotionStage.fVelocity;
        fTarAcc := -stMotionStage.fAcceleration;
    END_IF
ELSE
    fTarPos := fActPos;
    fTarVel := 0.0;
    fTarAcc := 0.0;
END_IF
END_METHOD


METHOD PUBLIC SetTargetPosVelAcc3D
VAR_INPUT
    stMotionStageX : ST_MotionStage;
    stMotionStageY : ST_MotionStage;
    stMotionStageZ : ST_MotionStage;
    fbActPosVec3 : FB_Vec3;
END_VAR
VAR_OUTPUT
    fbTarPosVec3 : FB_Vec3;
    fbTarVelVec3 : FB_Vec3;
    fbTarAccVec3 : FB_Vec3;
END_VAR
VAR
    fTarPosX : LREAL;
    fTarPosY : LREAL;
    fTarPosZ : LREAL;

    fTarVelX : LREAL;
    fTarVelY : LREAL;
    fTarVelZ : LREAL;

    fTarAccX : LREAL;
    fTarAccY : LREAL;
    fTarAccZ : LREAL;
END_VAR

SetTargetPosVelAcc1D(
    stMotionStage := stMotionStageX,
    fActPos := fbActPosVec3.x,
    fTarPos => fTarPosX,
    fTarVel => fTarVelX,
    fTarAcc => fTarAccX
);

SetTargetPosVelAcc1D(
    stMotionStage := stMotionStageY,
    fActPos := fbActPosVec3.y,
    fTarPos => fTarPosY,
    fTarVel => fTarVelY,
    fTarAcc => fTarAccY
);

SetTargetPosVelAcc1D(
    stMotionStage := stMotionStageZ,
    fActPos := fbActPosVec3.z,
    fTarPos => fTarPosZ,
    fTarVel => fTarVelZ,
    fTarAcc => fTarAccZ
);

fbTarPosVec3.Set(fTarPosX, fTarPosY, fTarPosZ);
fbTarVelVec3.Set(fTarVelX, fTarVelY, fTarVelZ);
fbTarAccVec3.Set(fTarAccX, fTarAccY, fTarAccZ);
END_METHOD

END_FUNCTION_BLOCK

// ---- Tests/FB_TestHelperSetAndMove_Test.TcPOU
FUNCTION_BLOCK FB_TestHelperSetAndMove_Test EXTENDS TcUnit.FB_TestSuite
(*
    Ensure that the test helper function block works as needed.
    Without this, all tests that need motion cannot pass.
*)
VAR
    stMotionStage: ST_MotionStage;
    fbMotionStage: FB_MotionStage;
    fbTestMove: FB_TestHelperSetAndMove;
    rtResetDone: R_TRIG;
    rtSetDone: R_TRIG;
    rtMotionStart: R_TRIG;
    rtMoveDone: R_TRIG;
END_VAR


fbMotionStage(stMotionStage:=stMotionstage);
BasicMotion();

METHOD PRIVATE BasicMotion
VAR_INPUT
END_VAR

TEST('BasicMotion');

IF NOT fbTestMove.bExecute THEN
    stMotionStage.bError := TRUE;
END_IF
fbTestMove(
    stMotionStage:=stMotionStage,
    bExecute:=TRUE,
    fStartPosition:=15.0,
    fGoalPosition:=17.0,
    fVelocity:=1.0,
    bHWEnable:=TRUE,
);
rtResetDone(CLK:=fbTestMove.bResetDone);
rtSetDone(CLK:=fbTestMove.bSetDone);
rtMotionStart(CLK:=fbTestMove.bMotionStarted);
rtMoveDone(CLK:=fbTestMove.bMoveDone);
IF rtResetDone.Q THEN
    AssertFalse(
        Condition:=stMotionStage.bError,
        Message:='Reset did not clear error',
    );
    AssertEquals_LREAL(
        Expected:=stMotionStage.stAxisStatus.fActPosition,
        Actual:=fbTestMove.fActPosition,
        Delta:=0,
        Message:='Real position output does not match real position.',
    );
END_IF
IF rtSetDone.Q THEN
    AssertEquals_LREAL(
        Expected:=fbTestMove.fStartPosition,
        Actual:=fbTestMove.fActPosition,
        Delta:=0,
        Message:='Was not set to start position after set done',
    );
END_IF
IF rtMotionStart.Q THEN
    AssertTrue(
        Condition:=stMotionStage.bBusy,
        Message:='stMotionStage is not busy, but motion is said to have started.',
    );
    AssertTrue(
        Condition:=fbTestMove.fActPosition > fbTestMove.fStartPosition,
        Message:='stMotionStage has not moved, but motion is said to have started.',
    );
END_IF
IF rtMoveDone.Q THEN
    AssertEquals_LREAL(
        Expected:=fbTestMove.fGoalPosition,
        Actual:=fbTestMove.fActPosition,
        Delta:=0.001,
        Message:='Did not reach destination at move done',
    );
END_IF
IF fbTestMove.bError OR fbTestMove.tElapsed > T#5s OR (fbTestMove.bResetDone AND fbTestMove.bSetDone AND fbTestMove.bMotionStarted AND fbTestMove.bMoveDone) THEN
    AssertFalse(
        Condition:=fbTestMove.bError,
        Message:='Error in fbTestMove',
    );
    AssertFalse(
        Condition:=fbTestMove.tElapsed > T#5s,
        Message:='Timeout in basic motion test',
    );
    TEST_FINISHED();
END_IF
END_METHOD

END_FUNCTION_BLOCK

// ---- Tests/FB_PositionStateRead_Test.TcPOU
FUNCTION_BLOCK FB_PositionStateRead_Test EXTENDS TcUnit.FB_TestSuite
(*
    Test that FB_PositionStateRead works exactly how it should
    according to its API during normal and failure states.
*)
VAR
    stMotionStage: ST_MotionStage;
    fbMotionStage: FB_MotionStage;
    astPositionState: ARRAY[1..GeneralConstants.MAX_STATES] OF ST_PositionState;
    afbInternal: ARRAY[1..3] OF FB_PositionStateInternal;
    stDummyPos: ST_PositionState;
    fbTestMove: FB_TestHelperSetAndMove;
    fbRead: FB_PositionStateRead;

    nTestCounter: UINT;
    bOneTestDone: BOOL;
    fTestStartPos: LREAL;
    tonTimer: TON;
    nIter: DINT;
    bStatesReady: BOOL;
END_VAR


astPositionState[1].sName := 'UNO';
astPositionState[1].fPosition := 10;
astPositionState[1].fDelta := 1;
astPositionState[1].bValid := TRUE;
astPositionState[1].bUseRawCounts := FALSE;

astPositionState[2].sName := 'DOS';
astPositionState[2].fPosition := 20;
astPositionState[2].fDelta := 1;
astPositionState[2].bValid := FALSE;
astPositionState[2].bUseRawCounts := FALSE;

astPositionState[3].sName := 'TRES';
astPositionState[3].fPosition := 30;
astPositionState[3].fDelta := 1;
astPositionState[3].bValid := TRUE;
astPositionState[3].bUseRawCounts := FALSE;

astPositionState[4].sName := 'QUATRO';
astPositionState[4].fPosition := 30;
astPositionState[4].fDelta := 1;
astPositionState[4].bValid := FALSE;
astPositionState[4].bUseRawCounts := FALSE;

bStatesReady := TRUE;
FOR nIter := 1 TO 4 DO
    afbInternal[nIter](
        stMotionStage:=stMotionStage,
        stPositionState:=astPositionState[nIter],
    );
    bStatesReady := bStatesReady AND astPositionState[nIter].bUpdated;
END_FOR
fbMotionStage(stMotionStage:=stMotionStage);

// At position 1 check
TestStaticPosition(
    nTestIndex:=0,
    sTestName:='AtPos1',
    fPosition:=astPositionState[1].fPosition + 0.2 * astPositionState[1].fDelta,
    bKnownState:=TRUE,
    bMovingState:=FALSE,
    nPositionIndex:=1,
    stCurrentPosition:=astPositionState[1],
);
// Outside the deltas check
TestStaticPosition(
    nTestIndex:=1,
    sTestName:='OutsidePos1Delta',
    fPosition:=astPositionState[1].fPosition + 2 * astPositionState[1].fDelta,
    bKnownState:=FALSE,
    bMovingState:=FALSE,
    nPositionIndex:=0,
    stCurrentPosition:=stDummyPos,
);
// At invalid state 2 check
TestStaticPosition(
    nTestIndex:=2,
    sTestName:='AtInvalidPos',
    fPosition:=astPositionState[2].fPosition,
    bKnownState:=FALSE,
    bMovingState:=FALSE,
    nPositionIndex:=0,
    stCurrentPosition:=stDummyPos,
);
// At position 3 check
TestStaticPosition(
    nTestIndex:=3,
    sTestName:='AtPos3',
    fPosition:=astPositionState[3].fPosition - 0.5 * astPositionState[3].fDelta,
    bKnownState:=TRUE,
    bMovingState:=FALSE,
    nPositionIndex:=3,
    stCurrentPosition:=astPositionState[3],
);
// At position 3 and moving within bounds check
TestMovingPosition(
    nTestIndex:=4,
    sTestName:='MovingAt3',
    fStartPosition:=astPositionState[3].fPosition,
    fGoalPosition:=astPositionState[3].fPosition + 0.9 * astPositionState[3].fDelta,
    fVelocity:=0.001,
    bKnownState:=TRUE,
    bMovingState:=FALSE,
    nPositionIndex:=3,
    stCurrentPosition:=astPositionState[3],
);
// At position 3 and moving away check
TestMovingPosition(
    nTestIndex:=5,
    sTestName:='MovingFrom3',
    fStartPosition:=astPositionState[3].fPosition,
    fGoalPosition:=astPositionState[3].fPosition + 100 * astPositionState[3].fDelta,
    fVelocity:=0.001,
    bKnownState:=FALSE,
    bMovingState:=TRUE,
    nPositionIndex:=0,
    stCurrentPosition:=stDummyPos,
);
TestDupe(nTestIndex:=6);

IF bOneTestDone THEN
    bOneTestDone := FALSE;
    nTestCounter := nTestCounter + 1;
    fbTestMove(
        stMotionStage:=stMotionStage,
        bExecute:=FALSE,
    );
END_IF

METHOD PRIVATE Asserts
VAR_INPUT
    tTimeout: TIME;
    bKnownState: BOOL;
    bMovingState: BOOL;
    nPositionIndex: DINT;
    stCurrentPosition: ST_PositionState;
END_VAR
VAR
    abExpected: ARRAY[1..GeneralConstants.MAX_STATES] OF BOOL;
END_VAR

fbRead(
    stMotionStage:=stMotionStage,
    astPositionState:=astPositionstate,
);

